   VAR
      s_FB_TimerOnOffDelay_Connected { ExternalAccessible := 'False'; ExternalVisible := 'False'; ExternalWritable := 'False'; S7_SetPoint := 'False'} : "FB_TimerOnOffDelay";
      sR_TRIG_LogOffRequest {InstructionName := 'R_TRIG'; LibVersion := '1.0'; ExternalAccessible := 'False'; ExternalVisible := 'False'; ExternalWritable := 'False'; S7_SetPoint := 'False'} : R_TRIG;   // Siemens "R_TRIG" - to prepare the rising edge trigger on "ix_LogOffRequest" signal
      sUDT_MessageArray { ExternalAccessible := 'False'; ExternalVisible := 'False'; ExternalWritable := 'False'; S7_SetPoint := 'False'} : "UDT_Message";   // Message character array
      sa_Status { ExternalAccessible := 'False'; ExternalVisible := 'False'; ExternalWritable := 'False'} : Struct   // Status structure
         FIFOStatus { ExternalAccessible := 'False'; ExternalVisible := 'False'; ExternalWritable := 'False'} : "UDT_FifoStatus";   // FIFO status structure
         FIFOError { ExternalAccessible := 'False'; ExternalVisible := 'False'; ExternalWritable := 'False'; S7_SetPoint := 'True'} : Bool;   // FIFO data buffer full
         FIFOWarning { ExternalAccessible := 'False'; ExternalVisible := 'False'; ExternalWritable := 'False'; S7_SetPoint := 'True'} : Bool;   // FIFO Warning
         InvalidMsgArraySize { ExternalAccessible := 'False'; ExternalVisible := 'False'; ExternalWritable := 'False'} : Bool;   // Invalig message array size
      END_STRUCT;
      ss_Message { ExternalAccessible := 'False'; ExternalVisible := 'False'; ExternalWritable := 'False'} : String;   // Message character string
      sui_MsgArrayElNr { ExternalAccessible := 'False'; ExternalVisible := 'False'; ExternalWritable := 'False'} : UInt;   // Invalid message array size
      si_MaxMsgLen { ExternalAccessible := 'False'; ExternalVisible := 'False'; ExternalWritable := 'False'} : Int;   // Maximum message length
      si_MsgLen { ExternalAccessible := 'False'; ExternalVisible := 'False'; ExternalWritable := 'False'} : Int;   // String character message length
   END_VAR

   VAR CONSTANT
      cc_NULL : Char := '$00';   // NULL sign
      cc_STX : Char := '$02';   // Start of the text
      cc_ETX : Char := '$03';   // End of the text
      cs_MessageLength : String := '0006';   // Legth of the message
      cs_LogOffRequest : String := 'LS';   // Message type
   END_VAR


BEGIN
	(*
	----------------------------------------------------------------------------------------

	Version history:
	Date        | Version   | Author        | Remark
	----------------------------------------------------------------------------------------
	24/05/2019  | 0.1       | L.Klar        | first release MHS TIA 15.1
	29/06/2021  | 1.0       | F.Baten       | first release MHS TIA 16.4
	08/11/2021  | 1.1       | M.Piela       | Interface changes
	05/04/2022  | 1.2       | K.Pokorski    | Review
	21/02/2023  | 4.0       | F.Baten       | 4.0 Release TIA 17.5
	*)

	REGION 1 – FIFO header status update

	    // Mode 'S' - FIFO register status update
	    "FC_Fifo"(ic_Mode := 'S',
	              qUDT_Status => #sa_Status.FIFOStatus,
	              qx_Error => #sa_Status.FIFOError,
	              qx_Warning => #sa_Status.FIFOWarning,
	              iqv_Data := #sUDT_MessageArray,
	              iqUDT_FifoHeader := #iqUDT_FifoHeader,
	              iqv_DataBuffer := #iqa_FifoData);

	END_REGION

	REGION 2 – Message preparation

	    #s_FB_TimerOnOffDelay_Connected(iudi_OnDelayTime := #i_UDT_Facility_PLC.SS,
	                                    iudi_OffDelayTime := 0,
	                                    ix_SignalToDelay := #ix_Connected AND NOT #ix_ConnectionAccepted);


	    #sR_TRIG_LogOffRequest(CLK := #ix_LogOffRequest OR #s_FB_TimerOnOffDelay_Connected.qx_DelayedSignal);

	    IF (NOT #iqUDT_FifoHeader.Status.Full)                 // FIFO isn't full
	    THEN

	        IF (#sR_TRIG_LogOffRequest.Q                       // Trigger message
	            AND NOT #sa_Status.FIFOError)                   // No FIFO error
	        THEN
	            REGION 2.1 – Message preparation

	                // Heartbeat message composing according to the structure: STX,00,06,LS,ETX
	                #ss_Message := CONCAT(IN1 := #cc_STX,             // Start of message
	                                      IN2 := #cs_MessageLength,            // message length
	                                      IN3 := #cs_LogOffRequest,     // Log-off request message
	                                      IN4 := #cc_ETX);              // End of message

	            END_REGION

	            REGION 2.2 – Maximum number of the message characters

	                #si_MaxMsgLen := "FC_GetNrOfArrayEl"(iv_Array := #sUDT_MessageArray.Character);

	            END_REGION

	            REGION 2.3 – Length of the complete message

	                #si_MsgLen := LEN(#ss_Message);

	            END_REGION

	            REGION 2.4 –  Message array size validation

	                #sa_Status.InvalidMsgArraySize := #si_MsgLen > #si_MaxMsgLen;

	            END_REGION

	            REGION 2.5 –  Message character string conversion to a message array of characters

	                IF (NOT #sa_Status.InvalidMsgArraySize)     // Message character array size is valid
	                THEN

	                    Strg_TO_Chars(Strg := #ss_Message,
	                                  pChars := 0,
	                                  Cnt => #sui_MsgArrayElNr,
	                                  Chars := #sUDT_MessageArray.Character);
	                END_IF;

	            END_REGION

	            REGION 2.6 – Clearing remaining characters in the message character array

	                IF (NOT #sa_Status.InvalidMsgArraySize)     // Message character array size is valid
	                THEN

	                    // Filling up not used message character array elements with '$00' (ASCII - 16#00)
	                    FILL_BLK(IN := #cc_NULL,
	                             COUNT := UINT_TO_ULINT(INT_TO_UINT(#si_MaxMsgLen) - #sui_MsgArrayElNr),
	                             OUT => #sUDT_MessageArray.Character[#sui_MsgArrayElNr]);

	                END_IF;

	            END_REGION

	            REGION 2.7 – Message write into a FIFO register

	                IF NOT #sa_Status.InvalidMsgArraySize // Message character array size is valid
	                THEN

	                    // Mode 'W' - Write FIFO record
	                    "FC_Fifo"(ic_Mode := 'W',
	                              qUDT_Status => #sa_Status.FIFOStatus,
	                              qx_Error => #sa_Status.FIFOError,
	                              qx_Warning => #sa_Status.FIFOWarning,
	                              iqv_Data := #sUDT_MessageArray,
	                              iqUDT_FifoHeader := #iqUDT_FifoHeader,
	                              iqv_DataBuffer := #iqa_FifoData);
	                END_IF;

	            END_REGION

	        END_IF;

	        // In case of FIFO full, the FIFO full error bit and FIFO collective error bit are set
	    ELSE

	        #sa_Status.FIFOError := TRUE;
	        #sa_Status.FIFOStatus.FifoFull := TRUE;

	    END_IF;

	END_REGION

	REGION Close connection

	    IF #iqUDT_FifoHeader.TotalEntriesStored = 0
	        AND (#ix_LogOffRequest OR #s_FB_TimerOnOffDelay_Connected.qx_DelayedSignal)
	    THEN
	        #iqx_Reconnect := TRUE;
	    END_IF;


	END_REGION


	REGION 3 - Writing output

	    #qx_Error := #sa_Status.InvalidMsgArraySize         // Invalid message array size
	    OR #sa_Status.FIFOError;                            // FIFO error

	END_REGION
END_FUNCTION_BLOCK

FUNCTION_BLOCK "FB_FedExPacketLengthMessage"
TITLE = FB_Heartbeat
{ S7_Optimized_Access := 'TRUE' }
AUTHOR : MHSE
FAMILY : UPS_SpecificCommunication
VERSION : 3.0
// ATTRIBUTES
// AUTO_NUMBER = True
// BLOCK_NUMBER = 80
// END_ATTRIBUTES
//Function block to send and monitor the UPS heartbeat message.
   VAR_INPUT
      iUDT_Facility { ExternalAccessible := 'False'; ExternalVisible := 'False'; ExternalWritable := 'False'} : "UDT_FedExFacility";   // System configuration
      is_LOConEquipment { ExternalAccessible := 'False'; ExternalVisible := 'False'; ExternalWritable := 'False'} : String[3];   // Location of the equipment
      is_DEPCOD { ExternalAccessible := 'False'; ExternalVisible := 'False'; ExternalWritable := 'False'} : String[6];   // Depot Code
      is_TYPofEquipment { ExternalAccessible := 'False'; ExternalVisible := 'False'; ExternalWritable := 'False'} : String[3];   // Type of equipment
      is_NumberOfTheEquipment { ExternalAccessible := 'False'; ExternalVisible := 'False'; ExternalWritable := 'False'} : String[3];   // Number of the equipment 001-999
      is_TrayCellNumber { ExternalAccessible := 'False'; ExternalVisible := 'False'; ExternalWritable := 'False'} : String[3];   // Tray/Cell number (for loop sorters) or generated by LLC (on line sorters).
      is_SorterNumber { ExternalAccessible := 'False'; ExternalVisible := 'False'; ExternalWritable := 'False'} : String[2];   // Sorter number
      is_InductionNumber { ExternalAccessible := 'False'; ExternalVisible := 'False'; ExternalWritable := 'False'} : String[2];   // Induction number
      is_AreaNumber { ExternalAccessible := 'False'; ExternalVisible := 'False'; ExternalWritable := 'False'} : String[2];   // Area number
      ii_Gin { ExternalAccessible := 'False'; ExternalVisible := 'False'; ExternalWritable := 'False'} : Int;   // GIN number
   END_VAR

   VAR_OUTPUT
      qx_Error { ExternalAccessible := 'False'; ExternalVisible := 'False'; ExternalWritable := 'False'} : Bool;   // Error
   END_VAR

   VAR_IN_OUT
      iqUDT_FifoHeader : "UDT_FifoHeader";   // FIFO header
      iqa_FifoData : Array[*] of "UDT_Message";   // FIFO data
      iqUDT_CustomerID : "UDT_FedExCustomerID";
   END_VAR

   VAR
      sFB_FedExCustomerID { ExternalAccessible := 'False'; ExternalVisible := 'False'; ExternalWritable := 'False'; S7_SetPoint := 'False'} : "FB_FedExCustomerID";
      sUDT_MessageArray { ExternalAccessible := 'False'; ExternalVisible := 'False'; ExternalWritable := 'False'; S7_SetPoint := 'False'} : "UDT_Message";   // Message character array
      sa_Status { ExternalAccessible := 'False'; ExternalVisible := 'False'; ExternalWritable := 'False'} : Struct   // Status structure
         FIFOStatus { ExternalAccessible := 'False'; ExternalVisible := 'False'; ExternalWritable := 'False'} : "UDT_FifoStatus";   // FIFO status structure
         FIFOError { ExternalAccessible := 'False'; ExternalVisible := 'False'; ExternalWritable := 'False'; S7_SetPoint := 'True'} : Bool;   // FIFO data buffer full
         FIFOWarning { ExternalAccessible := 'False'; ExternalVisible := 'False'; ExternalWritable := 'False'; S7_SetPoint := 'True'} : Bool;   // FIFO error
         InvalidGIN { ExternalAccessible := 'False'; ExternalVisible := 'False'; ExternalWritable := 'False'} : Bool;   //  Invalid GIN
         InvalidMessageLength { ExternalAccessible := 'False'; ExternalVisible := 'False'; ExternalWritable := 'False'} : Bool;   // Calculated message length is different than required
         InvalidMsgArraySize { ExternalAccessible := 'False'; ExternalVisible := 'False'; ExternalWritable := 'False'} : Bool;   // Length of the message is bigger than length of message array
      END_STRUCT;
      sa_Statistics { ExternalAccessible := 'False'; ExternalVisible := 'False'; ExternalWritable := 'False'} : Struct   // Statistics structure
         NotSentWrongMsgLen { ExternalAccessible := 'False'; ExternalVisible := 'False'; ExternalWritable := 'False'} : DInt;   // COMISSIONING PURPOSE Messages not sent because built message length does not match with required message length
      END_STRUCT;
      ss_LLCSystemID { ExternalAccessible := 'False'; ExternalVisible := 'False'; ExternalWritable := 'False'} : String[15];   // Identifier of Low-Level controls
      ss_SequencialID { ExternalAccessible := 'False'; ExternalVisible := 'False'; ExternalWritable := 'False'} : String[6];   // Identifier of Low-Level controls
      ss_Message { ExternalAccessible := 'False'; ExternalVisible := 'False'; ExternalWritable := 'False'} : String;   // Message character string
      ss_PackageID { ExternalAccessible := 'False'; ExternalVisible := 'False'; ExternalWritable := 'False'} : String;   // Identifier of Low-Level controls
      ss_LEN { ExternalAccessible := 'False'; ExternalVisible := 'False'; ExternalWritable := 'False'} : String;   // Length of message
      ss_Gap { ExternalAccessible := 'False'; ExternalVisible := 'False'; ExternalWritable := 'False'} : String;   // Parcel leading gap
      ss_GapUOM { ExternalAccessible := 'False'; ExternalVisible := 'False'; ExternalWritable := 'False'} : String;   // Gap units
      ss_Length { ExternalAccessible := 'False'; ExternalVisible := 'False'; ExternalWritable := 'False'} : String;   // Parcel length
      sui_MsgArrayElNr { ExternalAccessible := 'False'; ExternalVisible := 'False'; ExternalWritable := 'False'} : UInt;   // Message array size
      si_OldGin { ExternalAccessible := 'False'; ExternalVisible := 'False'; ExternalWritable := 'False'} : Int;   // Previous Gin
      si_StringLen { ExternalAccessible := 'False'; ExternalVisible := 'False'; ExternalWritable := 'False'} : Int;   // Length of string used in loops to pad string with spaces or 0
      si_LenFillLoop { ExternalAccessible := 'False'; ExternalVisible := 'False'; ExternalWritable := 'False'} : Int;   // Loop couter
      si_MaxMsgLen { ExternalAccessible := 'False'; ExternalVisible := 'False'; ExternalWritable := 'False'} : Int;   // Maximum message length
      si_MsgLen { ExternalAccessible := 'False'; ExternalVisible := 'False'; ExternalWritable := 'False'} : Int;   // String character message length
   END_VAR

   VAR CONSTANT
      cc_NULL : Char := '$00';   // NULL sign
      cc_STX : Char := '$02';   // Start of the text
      cc_ETX : Char := '$03';   // End of the text
      cs_Length : String := '0081';   // Legth of the message
      cs_MessageType : String := 'PL';   // Message type
   END_VAR


BEGIN
	(*
	----------------------------------------------------------------------------------------

	Version history:
	Date        | Version   | Author        | Remark
	----------------------------------------------------------------------------------------
	29/06/2021  | 1.0       | F.Baten       | first release MHS TIA 16.0
	10/11/2021  | 1.2       | M.Piela       | Updating regions numbering and interface changes
	05/04/2022  | 1.3       | K.Pokorski    | Review
	30/06/2022  | 1.4       | K.Pokorski    | Add cusotmer ID generation and swap GIN with Customer ID
	21/02/2023  | 4.0       | F.Baten       | 4.0 Release TIA 17.5
	*)

	REGION 1 – FIFO header status update

	    // Mode 'S' - FIFO register status update
	    "FC_Fifo"(ic_Mode := 'S',
	              qUDT_Status => #sa_Status.FIFOStatus,
	              qx_Error => #sa_Status.FIFOError,
	              qx_Warning => #sa_Status.FIFOWarning,
	              iqv_Data := #sUDT_MessageArray,
	              iqUDT_FifoHeader := #iqUDT_FifoHeader,
	              iqv_DataBuffer := #iqa_FifoData);
	END_REGION

	REGION 2 - GIN validation

	    // GIN validation
	    #sa_Status.InvalidGIN :=
	    #ii_Gin < 1
	    OR #ii_Gin > 9999;

	END_REGION

	REGION 3 – Message preparation

	    IF NOT #iqUDT_FifoHeader.Status.Full                 // FIFO isn't full
	    THEN
	        IF #ii_Gin <> #si_OldGin AND NOT #sa_Status.InvalidGIN

	        THEN
	            REGION 3.1 - Sequencial ID

	                // Assign CustomerID
	                #sFB_FedExCustomerID(ii_Gin := #ii_Gin,
	                                     iqUDT_CustomerID := #iqUDT_CustomerID);


	                // ss_SequencialID character string clearing
	                #ss_SequencialID := '';

	                // ss_SequencialID double integer input conversion to a character string
	                VAL_STRG(IN := "DB_GIN".GIN[#ii_Gin].FedEx.CustomerID,
	                         SIZE := 0,
	                         PREC := 0,
	                         FORMAT := 0,
	                         P := 1,
	                         OUT => #ss_SequencialID);
	                // Length of the ss_SequencialID character string
	                #si_StringLen := LEN(#ss_SequencialID);

	                // ss_SequencialID character string leading zeros addition
	                IF (#si_StringLen < 6)
	                THEN
	                    FOR #si_LenFillLoop := 1 TO 6 - #si_StringLen DO
	                        #ss_SequencialID := CONCAT(IN1 := '0',
	                                                   IN2 := #ss_SequencialID);
	                    END_FOR;
	                END_IF;
	            END_REGION

	            REGION 3.2 - LLC System ID
	                // Build LLC Syatem ID
	                #ss_LLCSystemID := CONCAT(IN1 := #is_DEPCOD,
	                                          IN2 := #is_LOConEquipment,
	                                          IN3 := #is_TYPofEquipment,
	                                          IN4 := #is_NumberOfTheEquipment);
	            END_REGION

	            REGION 3.3 - Package ID
	                // Build Package ID
	                #ss_PackageID := CONCAT(IN1 := #is_TrayCellNumber,
	                                        IN2 := #is_SorterNumber,
	                                        IN3 := #is_InductionNumber,
	                                        IN4 := #is_AreaNumber,
	                                        IN5 := #ss_SequencialID);
	            END_REGION

	            REGION 3.4 - Gap
	                // Gap character string clearing
	                #ss_Gap := '';

	                IF ("DB_GIN".GIN[#ii_Gin].General.LeadingGap > 999)
	                THEN
	                    #ss_Gap := '999';
	                ELSE

	                    // Gap integer input conversion to a character string
	                    VAL_STRG(IN := "DB_GIN".GIN[#ii_Gin].General.LeadingGap,
	                             SIZE := 0,
	                             PREC := 0,
	                             FORMAT := 0,
	                             P := 1,
	                             OUT => #ss_Gap);
	                    // Length of the gap character string
	                    #si_StringLen := LEN(#ss_Gap);
	                    // Gap character string leading zeros addition
	                    IF (#si_StringLen < 3)
	                    THEN
	                        FOR #si_LenFillLoop := 1 TO 3 - #si_StringLen DO
	                            #ss_Gap := CONCAT(IN1 := '0',
	                                              IN2 := #ss_Gap);
	                        END_FOR;
	                    END_IF;
	                END_IF;
	                #ss_GapUOM := 'CM';
	            END_REGION

	            REGION 3.5 - Length
	                // Length character string clearing
	                #ss_Length := '';
	                // Gap integer input conversion to a character string
	                VAL_STRG(IN := "DB_GIN".GIN[#ii_Gin].General.Length,
	                         SIZE := 0,
	                         PREC := 0,
	                         FORMAT := 0,
	                         P := 1,
	                         OUT => #ss_Length);
	                // Length of the gap character string
	                #si_StringLen := LEN(#ss_Length);
	                // Gap character string leading zeros addition
	                IF (#si_StringLen < 3)
	                THEN
	                    FOR #si_LenFillLoop := 1 TO 3 - #si_StringLen DO
	                        #ss_Length := CONCAT(IN1 := '0',
	                                             IN2 := #ss_Length);
	                    END_FOR;
	                END_IF;

	            END_REGION


	            REGION 3.6 – Message preparation
	                // Message composing according to the structure: STX,BODY ,ETX
	                #ss_Message := CONCAT(IN1 := #cc_STX,
	                                      IN2 := #cs_Length,
	                                      IN3 := #cs_MessageType,
	                                      IN4 := #ss_LLCSystemID,
	                                      IN5 := #ss_PackageID,
	                                      IN6 := "DB_GIN".GIN[#ii_Gin].FedEx.PackageEntrancePoint,
	                                      IN7 := "DB_GIN".GIN[#ii_Gin].FedEx.PackageEntranceState,
	                                      IN8 := #ss_Gap,
	                                      IN9 := #ss_Length,
	                                      IN10 := #ss_GapUOM,
	                                      IN11 := "DB_Time".Timestamp,
	                                      IN12 := #iUDT_Facility.TimeZoneDesignator,
	                                      IN13 := #cc_ETX);

	            END_REGION

	            REGION 3.7 – Maximum number of the message characters

	                #si_MaxMsgLen := "FC_GetNrOfArrayEl"(iv_Array := #sUDT_MessageArray.Character);

	            END_REGION

	            REGION 3.8 – Length of the complete message

	                #si_MsgLen := LEN(#ss_Message);

	                // Message length validation
	                #sa_Status.InvalidMessageLength := #si_MsgLen - 2 <> STRING_TO_INT(#cs_Length);

	            END_REGION

	            REGION 3.9 –  Message array size validation

	                #sa_Status.InvalidMsgArraySize := #si_MsgLen > #si_MaxMsgLen;

	            END_REGION

	            REGION 3.10 –  Message character string conversion to a message array of characters

	                IF (NOT #sa_Status.InvalidMsgArraySize)     // Message character array size is valid
	                THEN

	                    Strg_TO_Chars(Strg := #ss_Message,
	                                  pChars := 0,
	                                  Cnt => #sui_MsgArrayElNr,
	                                  Chars := #sUDT_MessageArray.Character);

	                END_IF;

	            END_REGION

	            REGION 3.11 – Clearing remaining characters in the message character array

	                IF (NOT #sa_Status.InvalidMsgArraySize)     // Message character array size is valid
	                THEN

	                    // Filling up not used message character array elements with '$00' (ASCII - 16#00)
	                    FILL_BLK(IN := #cc_NULL,
	                             COUNT := UINT_TO_ULINT(INT_TO_UINT(#si_MaxMsgLen) - #sui_MsgArrayElNr),
	                             OUT => #sUDT_MessageArray.Character[#sui_MsgArrayElNr]);

	                END_IF;

	            END_REGION

	            REGION 3.12 – Message write into a FIFO register

	                IF NOT #sa_Status.InvalidMsgArraySize          // Message character array size is valid
	                    AND NOT #sa_Status.InvalidMessageLength     // Message length size validation
	                THEN

	                    // Mode 'W' - Write FIFO record
	                    "FC_Fifo"(ic_Mode := 'W',
	                              qUDT_Status => #sa_Status.FIFOStatus,
	                              qx_Error => #sa_Status.FIFOError,
	                              qx_Warning => #sa_Status.FIFOWarning,
	                              iqv_Data := #sUDT_MessageArray,
	                              iqUDT_FifoHeader := #iqUDT_FifoHeader,
	                              iqv_DataBuffer := #iqa_FifoData);
	                ELSE
	                    // Increase counter messages not sent because of wrong message length
	                    #sa_Statistics.NotSentWrongMsgLen += 1;


	                END_IF;

	            END_REGION
	            #si_OldGin := #ii_Gin;
	        END_IF;
	        // In case of FIFO full, the FIFO full error bit and FIFO collective error bit are set
	    ELSE

	        #sa_Status.FIFOError := TRUE;
	        #sa_Status.FIFOStatus.FifoFull := TRUE;

	    END_IF;

	END_REGION

	REGION 4 - Writing outputs

	    #qx_Error := #sa_Status.InvalidMessageLength        // Invalid message length
	    OR #sa_Status.InvalidGIN                            // Invalid GIN
	    OR #sa_Status.InvalidMsgArraySize                   // Invalid message array size
	    OR #sa_Status.FIFOError;                            // FIFO error

	END_REGION
END_FUNCTION_BLOCK

FUNCTION_BLOCK "FB_FedExChute2Brakes1Stop"
{ S7_Optimized_Access := 'TRUE' }
VERSION : 0.1
// ATTRIBUTES
// AUTO_NUMBER = True
// BLOCK_NUMBER = 237
// END_ATTRIBUTES
   VAR_INPUT
      iUDT_ChuteConfiguration { ExternalAccessible := 'False'; ExternalVisible := 'False'; ExternalWritable := 'False'} : "UDT_Chute3BrakesConfiguration";   // Chute configuration structure
      iUDT_Facility { ExternalAccessible := 'False'; ExternalVisible := 'False'; ExternalWritable := 'False'} : "UDT_FedExFacility";   // System configuration
      ix_PECChuteFull { ExternalAccessible := 'False'; ExternalVisible := 'False'; ExternalWritable := 'False'} : Bool;   // TRUE when chute full photoye is not blocked
      ix_PECBrakeTop { ExternalAccessible := 'False'; ExternalVisible := 'False'; ExternalWritable := 'False'} : Bool;   // TRUE when first (Top) brake assembly photoye is not blocked
      ix_PECBrakeMiddle { ExternalAccessible := 'False'; ExternalVisible := 'False'; ExternalWritable := 'False'} : Bool;   // TRUE when second (Middle) brake assembly photoye is not blocked
      ix_PECBrakeBottom { ExternalAccessible := 'False'; ExternalVisible := 'False'; ExternalWritable := 'False'} : Bool;   // TRUE when third (End Stop) brake assembly photoye is not blocked
      ix_PECStopTop { ExternalAccessible := 'False'; ExternalVisible := 'False'; ExternalWritable := 'False'} : Bool;   // TRUE when first/Top brake assembly photoye is not blocked
      ix_PECStopMiddle { ExternalAccessible := 'False'; ExternalVisible := 'False'; ExternalWritable := 'False'} : Bool;   // TRUE when second/Middle brake assembly photoye is not blocked
      ix_PECStopBottom { ExternalAccessible := 'False'; ExternalVisible := 'False'; ExternalWritable := 'False'} : Bool;   // TRUE when third/(End Stop) brake assembly photoye is not blocked
      ix_ChuteJam { ExternalAccessible := 'False'; ExternalVisible := 'False'; ExternalWritable := 'False'} : Bool;   // TRUE when external jam appear
      ix_SafetyOk { ExternalAccessible := 'False'; ExternalVisible := 'False'; ExternalWritable := 'False'} : Bool;   // TRUE when safety is ok
      ix_HardwareOk { ExternalAccessible := 'False'; ExternalVisible := 'False'; ExternalWritable := 'False'} : Bool;   // TRUE when hardware is ok
      ix_EnergySave { ExternalAccessible := 'False'; ExternalVisible := 'False'; ExternalWritable := 'False'} : Bool;   // TRUE when enery save is active
   END_VAR

   VAR_OUTPUT
      qUDT_HMIStatus { ExternalAccessible := 'False'; ExternalVisible := 'False'; ExternalWritable := 'False'} : "UDT_Chute3BrakeStatus";   // HMI status structure
      qUDT_Status { ExternalAccessible := 'False'; ExternalVisible := 'False'; ExternalWritable := 'False'} : "UDT_CommonStatus";   // Common status structure
      qUDT_StatusToXBS { ExternalAccessible := 'False'; ExternalVisible := 'False'; ExternalWritable := 'False'} : "UDT_XBSChuteInterfaceSend";
      qx_Lamp { ExternalAccessible := 'False'; ExternalVisible := 'False'; ExternalWritable := 'False'} : Bool;   // Chute Lamp Jam/Full
      qx_BrakeValve1 { ExternalAccessible := 'False'; ExternalVisible := 'False'; ExternalWritable := 'False'} : Bool;   // First brake valve assembly
      qx_BrakeValve2 { ExternalAccessible := 'False'; ExternalVisible := 'False'; ExternalWritable := 'False'} : Bool;   // Second brake valve  assembly
      qx_BrakeValve3 { ExternalAccessible := 'False'; ExternalVisible := 'False'; ExternalWritable := 'False'} : Bool;   // Third brake valve assembly
   END_VAR

   VAR_IN_OUT
      iqUDT_EquipmentControl : "UDT_EquipmentControl";   // Equipment control structure
      iqUDT_Statistics : "UDT_Chute3BrakeStatistics";   // Statistics structure
      iqUDT_HandShake : "UDT_ConveyorHandshake";   // Downstream handshake structure
      iqUDT_HandShakeUp : "UDT_ConveyorHandshake";   // Upstream handshake structure
      iqUDT_ChuteCommand : "UDT_Chute3BrakeCommand";   // Command strucutre
      iqUDT_FifoHighPriorityHLC : "UDT_FifoHeader";   // FIFO UDS send Header
      iqa_FifoHighPriorityHLC : Array[*] of "UDT_Message";   // FIFO UDS send data
   END_VAR

   VAR
      sUDT_CommonStatus { ExternalAccessible := 'False'; ExternalVisible := 'False'; ExternalWritable := 'False'; S7_SetPoint := 'False'} : "UDT_CommonStatus";   // Common status structure
      sUDT_CommonStatusOld { ExternalAccessible := 'False'; ExternalVisible := 'False'; ExternalWritable := 'False'; S7_SetPoint := 'False'} : "UDT_CommonStatus";   // Auxiliary status structure
      sUDT_HMIStatus { ExternalAccessible := 'False'; ExternalVisible := 'False'; ExternalWritable := 'False'; S7_SetPoint := 'False'} : "UDT_Chute3BrakeStatus";   // HMI status structure
      sUDT_Configuration { ExternalAccessible := 'False'; ExternalVisible := 'False'; ExternalWritable := 'False'; S7_SetPoint := 'False'} : "UDT_Chute3BrakesConfiguration";   // Auxiliary equipment control structure
      sFB_PneumaticBrakeUnitAssemby1 { ExternalAccessible := 'False'; ExternalVisible := 'False'; ExternalWritable := 'False'; S7_SetPoint := 'False'} : "FB_PneumaticBrakeUnit";   // Function to control a first pneumatic brake contol
      sFB_PneumaticBrakeUnitAssemby2 { ExternalAccessible := 'False'; ExternalVisible := 'False'; ExternalWritable := 'False'; S7_SetPoint := 'False'} : "FB_PneumaticBrakeUnit";   // Function to control a secound pneumatic brake contol
      sFB_StopRoller { ExternalAccessible := 'False'; ExternalVisible := 'False'; ExternalWritable := 'False'; S7_SetPoint := 'False'} : "FB_StopRoller";   // Function to control stoping of the roller
      sFB_FedExEquipmentStatusMessage { ExternalAccessible := 'False'; ExternalVisible := 'False'; ExternalWritable := 'False'; S7_SetPoint := 'False'} : "FB_FedExEquipmentStatusMessage";   // Equipment status structure message
      sFB_TimerOnOffDelayPECFul { ExternalAccessible := 'False'; ExternalVisible := 'False'; ExternalWritable := 'False'; S7_SetPoint := 'False'} : "FB_TimerOnOffDelay";   // Filtering full photo eye signal
      sFB_TimerOnOffDelayPECHalfFull { ExternalAccessible := 'False'; ExternalVisible := 'False'; ExternalWritable := 'False'; S7_SetPoint := 'False'} : "FB_TimerOnOffDelay";   // Filtering half full photo eye signal
      sFB_TimerOnOffDelayPECMiddle { ExternalAccessible := 'False'; ExternalVisible := 'False'; ExternalWritable := 'False'; S7_SetPoint := 'False'} : "FB_TimerOnOffDelay";   // Filtering middle photo eye signal
      sFB_TimerOnOffDelayStopRollerLongBrakePause { ExternalAccessible := 'False'; ExternalVisible := 'False'; ExternalWritable := 'False'; S7_SetPoint := 'False'} : "FB_TimerOnOffDelay";   // Filtering common signal from all signals needed to increase brake pause
      sR_TRIG_ChuteFull {InstructionName := 'R_TRIG'; LibVersion := '1.0'; ExternalAccessible := 'False'; ExternalVisible := 'False'; ExternalWritable := 'False'; S7_SetPoint := 'False'} : R_TRIG;   // Rising edge to chute full
      sR_TRIG_ChuteJam {InstructionName := 'R_TRIG'; LibVersion := '1.0'; ExternalAccessible := 'False'; ExternalVisible := 'False'; ExternalWritable := 'False'; S7_SetPoint := 'False'} : R_TRIG;   // Rising edge to chute jam
      sR_TRIG_ChuteHalfFull {InstructionName := 'R_TRIG'; LibVersion := '1.0'; ExternalAccessible := 'False'; ExternalVisible := 'False'; ExternalWritable := 'False'; S7_SetPoint := 'False'} : R_TRIG;   // Rising edge to chute half full
      sR_TRIG_DisableFromHMI {InstructionName := 'R_TRIG'; LibVersion := '1.0'; ExternalAccessible := 'False'; ExternalVisible := 'False'; ExternalWritable := 'False'; S7_SetPoint := 'False'} : R_TRIG;   // Rising edge to disable chute from HMI
      sR_TRIG_DisableFromHLC {InstructionName := 'R_TRIG'; LibVersion := '1.0'; ExternalAccessible := 'False'; ExternalVisible := 'False'; ExternalWritable := 'False'; S7_SetPoint := 'False'} : R_TRIG;   // Rising edge to disable chute from HLC
      sF_TRIG_UpdateStatus {InstructionName := 'F_TRIG'; LibVersion := '1.0'; ExternalAccessible := 'False'; ExternalVisible := 'False'; ExternalWritable := 'False'; S7_SetPoint := 'False'} : F_TRIG;
      ss_StatusCode { ExternalAccessible := 'False'; ExternalVisible := 'False'; ExternalWritable := 'False'} : String[3];   // Status code
      sx_MasterValve { ExternalAccessible := 'False'; ExternalVisible := 'False'; ExternalWritable := 'False'} : Bool;   // Master valve
      sx_StopActive1 { ExternalAccessible := 'False'; ExternalVisible := 'False'; ExternalWritable := 'False'} : Bool;   // First brake valve assembly is active
      sx_StopActive2 { ExternalAccessible := 'False'; ExternalVisible := 'False'; ExternalWritable := 'False'} : Bool;   // Second brake valve assembly is active
      sx_StopActive3 { ExternalAccessible := 'False'; ExternalVisible := 'False'; ExternalWritable := 'False'} : Bool;   // Third brake valve assembly is active
      sx_PECFullFiltered { ExternalAccessible := 'False'; ExternalVisible := 'False'; ExternalWritable := 'False'} : Bool;   // Delayed full photo eye signal
      sx_PECHalfFullFiltered { ExternalAccessible := 'False'; ExternalVisible := 'False'; ExternalWritable := 'False'} : Bool;   // Delayed half full photo eye signal
      sx_PECMiddleFullFiltered { ExternalAccessible := 'False'; ExternalVisible := 'False'; ExternalWritable := 'False'} : Bool;   // Delayed middle full photo eye signal
      sx_StopRollerLongBrakePauseDelayed { ExternalAccessible := 'False'; ExternalVisible := 'False'; ExternalWritable := 'False'} : Bool;   // Delayed common signal from all signals needed to increase brake pause
      sx_StopRollerLongBrakePause { ExternalAccessible := 'False'; ExternalVisible := 'False'; ExternalWritable := 'False'} : Bool;   // Common signal from all signals needed to increase brake pause
      sx_ChuteFull { ExternalAccessible := 'False'; ExternalVisible := 'False'; ExternalWritable := 'False'} : Bool;   // Full status
      sx_ChuateHalfFull { ExternalAccessible := 'False'; ExternalVisible := 'False'; ExternalWritable := 'False'} : Bool;   // Half full occupation status
      sx_ChuteJam { ExternalAccessible := 'False'; ExternalVisible := 'False'; ExternalWritable := 'False'} : Bool;   // Jam status
      sx_MessageError { ExternalAccessible := 'False'; ExternalVisible := 'False'; ExternalWritable := 'False'} : Bool;   // Message error
   END_VAR


BEGIN
	(*
	----------------------------------------------------------------------------------------

	Version history:
	Date        | Version   | Author        | Remark
	----------------------------------------------------------------------------------------
	23/06/2021  | 0.0       | F. Baten      | first release TIA 15.1
	20/10/2021  | 0.1       | M. Piela      | Add statuses and statistics. Stylistic correction
	21/10/2021  | 0.2       | M. Piela      | Change brake stopper pause based on all pec delayed signal
	02/02/2022  | 0.3       | M. Piela      | Add Equipment status message
	22/02/2022  | 0.4       | M. Piela      | Update HMI Status
	04/04/2022  | 0.5       | S. Deulkar    | Updated status for XBS sorter
	25/06/2022  | 0.6       | M. Kurpiers   | Interface update
	25/06/2022  | 0.7       | M. Piela      | #sx_MasterValve inverted to top brake
	19/07/2022  | 0.8       | M. Piela      | Add external chute jam to the status
	21/02/2023  | 4.0       | F.Baten       | 4.0 Release TIA 17.5
	 *)

	REGION 1 - Write input status

	    IF #ix_HardwareOk
	    THEN
	        #sUDT_HMIStatus.Specific.DisableFromHMI := #iqUDT_ChuteCommand.DisableFromHMI;
	        #sUDT_HMIStatus.Specific.DisableFromHLC := #iqUDT_ChuteCommand.DisableFromHLC;
	        #sUDT_HMIStatus.Specific.ChuteFull := #sx_ChuteFull;
	        #sUDT_HMIStatus.Specific.ChuteHalfFull := #sx_ChuateHalfFull;
	        #sUDT_HMIStatus.Specific.ChuteJam := #sx_ChuteJam OR #ix_ChuteJam;
	        #sUDT_HMIStatus.Specific.BrakeFaultTop := FALSE;
	        #sUDT_HMIStatus.Specific.BrakeFaultMiddle := FALSE;
	        #sUDT_HMIStatus.Specific.BrakeFaultBottom := FALSE;
	    END_IF;

	END_REGION

	REGION 2 - Triggers

	    // Rising edge trigger full PEC status
	    #sR_TRIG_ChuteFull(CLK := #sx_ChuteFull);

	    // Rissing edge trigger jam PEC status
	    #sR_TRIG_ChuteJam(CLK := #sx_ChuteJam);

	    // Rissing edge trigger hafl full PEC status
	    #sR_TRIG_ChuteHalfFull(CLK := #sx_ChuateHalfFull);

	    // Rising edge trigger disable from HMI
	    #sR_TRIG_DisableFromHMI(CLK := #sUDT_HMIStatus.Specific.DisableFromHMI);

	    // Rising edge trigger disable from MFC
	    #sR_TRIG_DisableFromHLC(CLK := #sUDT_HMIStatus.Specific.DisableFromHLC);

	END_REGION

	REGION 3 - Timers

	    // Filtering full photo eye signal
	    #sFB_TimerOnOffDelayPECFul(iudi_OnDelayTime := #iUDT_ChuteConfiguration.PECFullOnDelay,
	                               iudi_OffDelayTime := #iUDT_ChuteConfiguration.PECFullOffDelay,
	                               ix_SignalToDelay := #ix_PECChuteFull,
	                               ix_Enable := TRUE,
	                               qx_DelayedSignal => #sx_PECFullFiltered);

	    //Filtering Half full photo eye signal
	    #sFB_TimerOnOffDelayPECHalfFull(iudi_OnDelayTime := #iUDT_ChuteConfiguration.PECHalfFullOnDelay,
	                                    iudi_OffDelayTime := #iUDT_ChuteConfiguration.PECHalfFullOffDelay,
	                                    ix_SignalToDelay := #ix_PECStopTop,
	                                    ix_Enable := TRUE,
	                                    qx_DelayedSignal => #sx_PECHalfFullFiltered);

	    //Filtering middle photo eye signal
	    #sFB_TimerOnOffDelayPECMiddle(iudi_OnDelayTime := #iUDT_ChuteConfiguration.PECMiddleOnDelay,
	                                  iudi_OffDelayTime := #iUDT_ChuteConfiguration.PECMiddleOffDelay,
	                                  ix_SignalToDelay := #ix_PECStopMiddle,
	                                  ix_Enable := TRUE,
	                                  qx_DelayedSignal => #sx_PECMiddleFullFiltered);

	    // Create common signal from all signals needed to increase brake pause
	    #sx_StopRollerLongBrakePause := #ix_PECBrakeMiddle
	    AND #ix_PECStopMiddle
	    AND #iqUDT_HandShake.RTR;     // Downstream conveyor is running

	    //Filtering common signal from all signals needed to increase brake pause
	    #sFB_TimerOnOffDelayStopRollerLongBrakePause(iudi_OnDelayTime := #iUDT_ChuteConfiguration.LongBrakePauseOnDelay,
	                                                 ix_SignalToDelay := #sx_StopRollerLongBrakePause,
	                                                 ix_Enable := TRUE,
	                                                 qx_DelayedSignal => #sx_StopRollerLongBrakePauseDelayed);

	END_REGION

	REGION 4 - Brake assembly

	    // Control first pneumatic break unit assembly
	    #sFB_PneumaticBrakeUnitAssemby1(iUDT_PneumaticBreakConfiguration := #iUDT_ChuteConfiguration.BrakeConfiguration1,
	                                    ix_PECBrake := #ix_PECBrakeTop,
	                                    ix_PECStop := #ix_PECStopTop,
	                                    ix_PECdownstream := #ix_PECBrakeMiddle,
	                                    ix_DownstreamStopActive := #sx_StopActive2,
	                                    ix_MasterValve := NOT #sx_MasterValve,
	                                    ix_SafetyOk := #ix_SafetyOk,
	                                    qx_Valve => #qx_BrakeValve1,
	                                    qx_StopActive => #sx_StopActive1,
	                                    iqUDT_EquipmentControl := #iqUDT_EquipmentControl);

	    // Control secound pneumatic break unit assembly
	    #sFB_PneumaticBrakeUnitAssemby2(iUDT_PneumaticBreakConfiguration := #iUDT_ChuteConfiguration.BrakeConfiguration2,
	                                    ix_PECBrake := #ix_PECBrakeMiddle,
	                                    ix_PECStop := #ix_PECStopMiddle,
	                                    ix_PECdownstream := #ix_PECBrakeBottom,
	                                    ix_DownstreamStopActive := #sx_StopActive3,
	                                    ix_SafetyOk := #ix_SafetyOk,
	                                    qx_Valve => #sx_MasterValve,
	                                    qx_StopActive => #sx_StopActive2,
	                                    iqUDT_EquipmentControl := #iqUDT_EquipmentControl);

	    // Control stop roller section
	    #sFB_StopRoller(iUDT_StopRollerConfiguration := #iUDT_ChuteConfiguration.StopperConfiguration,
	                    ix_Pressure := #ix_PECStopMiddle,
	                    ix_PECBrake := #ix_PECBrakeBottom,
	                    ix_PECStop := #ix_PECStopBottom,
	                    ix_DownstreamStopActive := NOT #iqUDT_HandShake.RTR,
	                    ix_SafetyOk := #ix_SafetyOk,
	                    ix_BrakePauseLong := #sx_StopRollerLongBrakePauseDelayed,
	                    qx_Valve => #qx_BrakeValve3,
	                    qx_StopActive => #sx_StopActive3,
	                    iqUDT_EquipmentControl := #iqUDT_EquipmentControl);

	    #qx_BrakeValve2 := #sx_MasterValve;

	END_REGION

	REGION 5 - Filling level

	    //Half full
	    IF NOT #sx_PECMiddleFullFiltered AND NOT #sx_PECHalfFullFiltered
	    THEN
	        #sx_ChuateHalfFull := TRUE;
	    END_IF;
	    IF #sx_PECMiddleFullFiltered AND #sx_PECHalfFullFiltered
	    THEN
	        #sx_ChuateHalfFull := FALSE;
	    END_IF;

	    //Full
	    IF NOT #sx_PECHalfFullFiltered AND NOT #"sx_PECFullFiltered"
	    THEN
	        #sx_ChuteFull := TRUE;
	    END_IF;
	    IF #sx_PECHalfFullFiltered AND #"sx_PECFullFiltered"
	    THEN
	        #sx_ChuteFull := FALSE;
	    END_IF;

	    // Jam
	    #sx_ChuteJam := #sx_PECHalfFullFiltered AND NOT #"sx_PECFullFiltered";

	END_REGION

	REGION 6 - Output

	    //Lamp signal enable
	    #qx_Lamp := NOT (#ix_ChuteJam OR #sx_ChuteJam) AND ((#sx_ChuteFull)
	    OR (#sx_ChuateHalfFull AND "DB_Memory"."Clock_1Hz"))
	    OR (#ix_ChuteJam OR #sx_ChuteJam) AND "DB_Memory"."Clock_2Hz";

	    //Send RTR signal to the sorter
	    #iqUDT_HandShakeUp.RTR := #ix_SafetyOk AND NOT (#ix_ChuteJam OR #sx_ChuteFull)
	    AND NOT #iqUDT_ChuteCommand.DisableFromHMI
	    AND NOT #iqUDT_ChuteCommand.DisableFromHLC;

	END_REGION

	REGION 7 - Statistics

	    // Chute disable from HMI.
	    IF #sUDT_HMIStatus.Specific.DisableFromHMI
	        OR #iqUDT_EquipmentControl.Command.ResetData
	    THEN
	        "FC_Statistics"(ix_Reset := #iqUDT_EquipmentControl.Command.ResetData,
	                        ix_Activate := #sUDT_HMIStatus.Specific.DisableFromHMI,
	                        ix_RTrigActivate := #sR_TRIG_DisableFromHMI.Q,
	                        iqUDT_Statistics := #iqUDT_Statistics.DisableFromHMI);
	    END_IF;

	    // Chute disable from HLC
	    IF #sUDT_HMIStatus.Specific.DisableFromHLC
	        OR #iqUDT_EquipmentControl.Command.ResetData
	    THEN
	        "FC_Statistics"(ix_Reset := #iqUDT_EquipmentControl.Command.ResetData,
	                        ix_Activate := #sUDT_HMIStatus.Specific.DisableFromHLC,
	                        ix_RTrigActivate := #sR_TRIG_DisableFromHLC.Q,
	                        iqUDT_Statistics := #iqUDT_Statistics.DisableFromHLC);
	    END_IF;

	    //Chute full
	    IF #sUDT_HMIStatus.Specific.ChuteFull
	        OR #iqUDT_EquipmentControl.Command.ResetData
	    THEN

	        "FC_Statistics"(ix_Reset := #iqUDT_EquipmentControl.Command.ResetData,
	                        ix_Activate := #sUDT_HMIStatus.Specific.ChuteFull,
	                        ix_RTrigActivate := #sR_TRIG_ChuteFull.Q,
	                        iqUDT_Statistics := #iqUDT_Statistics.ChuteFull);

	    END_IF;

	    //Chute half full
	    IF #sUDT_HMIStatus.Specific.ChuteHalfFull
	        OR #iqUDT_EquipmentControl.Command.ResetData
	    THEN

	        "FC_Statistics"(ix_Reset := #iqUDT_EquipmentControl.Command.ResetData,
	                        ix_Activate := #sUDT_HMIStatus.Specific.ChuteHalfFull,
	                        ix_RTrigActivate := #sR_TRIG_ChuteHalfFull.Q,
	                        iqUDT_Statistics := #iqUDT_Statistics.ChuteHalfFull);

	    END_IF;

	    //Chute jam
	    IF #sUDT_HMIStatus.Specific.ChuteJam
	        OR #iqUDT_EquipmentControl.Command.ResetData
	    THEN

	        "FC_Statistics"(ix_Reset := #iqUDT_EquipmentControl.Command.ResetData,
	                        ix_Activate := #sUDT_HMIStatus.Specific.ChuteJam,
	                        ix_RTrigActivate := #sR_TRIG_ChuteJam.Q,
	                        iqUDT_Statistics := #iqUDT_Statistics.ChuteJam);

	    END_IF;

	END_REGION

	REGION 8 - Status

	    //Error active
	    #sUDT_CommonStatus.Error := NOT #ix_HardwareOk OR NOT #ix_SafetyOk OR #sx_ChuteJam;

	    //Automation ON
	    #sUDT_CommonStatus.AutoON := #iqUDT_EquipmentControl.Command.AutomaticOn;

	    // Energy save active
	    #sUDT_CommonStatus.EnergySave := #ix_EnergySave;

	    // Running
	    #sUDT_CommonStatus.Running := #sUDT_CommonStatus.AutoON AND NOT #sUDT_CommonStatus.Error;

	    // Stopped
	    #sUDT_CommonStatus.Stopped := NOT #sUDT_CommonStatus.AutoON OR #sUDT_CommonStatus.Error;

	    // Safety not ok
	    #sUDT_CommonStatus.SafetyStop := NOT #ix_SafetyOk;

	    // Chute disabled
	    IF #sUDT_HMIStatus.Specific.DisableFromHMI OR #sUDT_HMIStatus.Specific.DisableFromHLC AND NOT #sUDT_CommonStatus.SafetyStop
	    THEN
	        #sUDT_HMIStatus.Status := "DB_HMIStatusConfiguration".DisableByManagement;
	    END_IF;

	    // Chute Half Full
	    IF #sUDT_HMIStatus.Specific.ChuteHalfFull AND NOT #sUDT_CommonStatus.SafetyStop
	    THEN
	        #sUDT_HMIStatus.Status := "DB_HMIStatusConfiguration".ChuteHalfFull;
	    END_IF;

	    //Chute Full
	    IF #sUDT_HMIStatus.Specific.ChuteFull AND NOT #sUDT_CommonStatus.SafetyStop
	    THEN
	        #sUDT_HMIStatus.Status := "DB_HMIStatusConfiguration".ChuteFull;
	    END_IF;

	    //Chute Jam
	    IF #sUDT_HMIStatus.Specific.ChuteJam AND NOT #sUDT_CommonStatus.SafetyStop
	    THEN
	        #sUDT_HMIStatus.Status := "DB_HMIStatusConfiguration".PECJam;
	    END_IF;

	    //Collecting F_TRIG on chute full, half full, jam or chute disabled status to update common status
	    #sF_TRIG_UpdateStatus(CLK := #sUDT_HMIStatus.Specific.ChuteHalfFull OR #sUDT_HMIStatus.Specific.ChuteFull
	                          OR #sUDT_HMIStatus.Specific.ChuteJam OR #sUDT_HMIStatus.Specific.DisableFromHMI
	                          OR #sUDT_HMIStatus.Specific.DisableFromHLC);

	    // HMI status update
	    IF #sUDT_CommonStatusOld <> #sUDT_CommonStatus OR #sF_TRIG_UpdateStatus.Q  // update on change
	    THEN
	        // HMI status initialization
	        #sUDT_HMIStatus.Status := 0;

	        // Energy save
	        IF #sUDT_CommonStatus.EnergySave
	        THEN
	            #sUDT_HMIStatus.Status := "DB_HMIStatusConfiguration".EnergySave;
	        END_IF;

	        // Running
	        IF #sUDT_CommonStatus.Running
	        THEN
	            #sUDT_HMIStatus.Status := "DB_HMIStatusConfiguration".Running;
	        END_IF;

	        // Stopped
	        IF #sUDT_CommonStatus.Stopped
	        THEN
	            #sUDT_HMIStatus.Status := "DB_HMIStatusConfiguration".Stopped;
	        END_IF;

	        // Error
	        IF #sUDT_CommonStatus.Error
	        THEN
	            #sUDT_HMIStatus.Status := "DB_HMIStatusConfiguration".Stopped;
	        END_IF;

	        // Safety stop
	        IF #sUDT_CommonStatus.SafetyStop
	        THEN
	            #sUDT_HMIStatus.Status := "DB_HMIStatusConfiguration".SafetyStop;
	        END_IF;

	        #sUDT_CommonStatusOld := #sUDT_CommonStatus;              // Copy status to memory
	        #qUDT_Status := #sUDT_CommonStatus;                       // Copy status to output

	    END_IF;

	    // Copy HMI status to output
	    #qUDT_HMIStatus := #sUDT_HMIStatus;

	END_REGION

	REGION 9 - Report to control block

	    // Function to manage report between control block and conveyor block
	    "FC_EquipmentReport"(iUDT_Status := #sUDT_CommonStatus,
	                         iqUDT_Control := #iqUDT_EquipmentControl);

	END_REGION

	REGION 10 - Equipment staus message

	    IF NOT #iqUDT_EquipmentControl.Command.AutomaticOn
	    THEN
	        #ss_StatusCode := '006'; //Inactive
	    ELSIF #sx_ChuteJam
	    THEN
	        #ss_StatusCode := '002';  //Chute Jam
	    ELSIF #sx_ChuteFull
	    THEN
	        #ss_StatusCode := '003';  // Chute Full
	    ELSIF #sx_ChuateHalfFull
	    THEN
	        #ss_StatusCode := '004';  // Chute Half full
	    ELSIF #iqUDT_ChuteCommand.DisableFromHMI OR #iqUDT_ChuteCommand.DisableFromHLC
	    THEN
	        #ss_StatusCode := '005'; // Chute Disabled
	    ELSE
	        #ss_StatusCode := '001'; //Chute is Clear
	    END_IF;

	    #sFB_FedExEquipmentStatusMessage(iUDT_Facility := #iUDT_Facility,
	                                     is_LOConEquipment := #iUDT_ChuteConfiguration.LOConEquipment, // Sorter number
	                                     is_DEPCOD := #iUDT_ChuteConfiguration.DEPCOD,
	                                     is_TYPofEquipment := 'PLC',
	                                     is_NumberOfTheEquipment := #iUDT_ChuteConfiguration.NumberOfTheEquipment,// PLC number
	                                     is_DeviceType := 'CHUTES',
	                                     is_DeviceID := #iUDT_ChuteConfiguration."Device ID", //Chute number
	                                     is_StatusCode := #ss_StatusCode,
	                                     qx_Error => #sx_MessageError,
	                                     iqUDT_FifoHeader := #iqUDT_FifoHighPriorityHLC,
	                                     iqa_FifoData := #iqa_FifoHighPriorityHLC);

	END_REGION

	REGION 11 XBS interface
	    // Map chute status to sorter
	    #qUDT_StatusToXBS.Full := #sUDT_HMIStatus.Specific.ChuteFull;
	    #qUDT_StatusToXBS.HalfFull := #sUDT_HMIStatus.Specific.ChuteHalfFull;
	    #qUDT_StatusToXBS.ReadyToReceive := NOT #sUDT_CommonStatus.Error AND #sUDT_CommonStatus.AutoON;
	    #qUDT_StatusToXBS.Running := #sUDT_CommonStatus.Running;
	    #qUDT_StatusToXBS.Fault := #sUDT_CommonStatus.Error;
	    #qUDT_StatusToXBS.Warning := #sUDT_CommonStatus.Warning;
	END_REGION

END_FUNCTION_BLOCK

FUNCTION_BLOCK "FB_FedExPolisorterGlobalEquipmentStatus"
{ S7_Optimized_Access := 'TRUE' }
VERSION : 0.1
// ATTRIBUTES
// AUTO_NUMBER = True
// BLOCK_NUMBER = 81
// END_ATTRIBUTES
   VAR_INPUT
      iUDT_FedExFacility { ExternalAccessible := 'False'; ExternalVisible := 'False'; ExternalWritable := 'False'} : "UDT_FedExFacility";   // System configuration
      is_LOConEquipment { ExternalAccessible := 'False'; ExternalVisible := 'False'; ExternalWritable := 'False'} : String[3];   // Location of the equipment
      is_DEPCOD { ExternalAccessible := 'False'; ExternalVisible := 'False'; ExternalWritable := 'False'} : String[6];   // Depot Code
      is_TYPofEquipment { ExternalAccessible := 'False'; ExternalVisible := 'False'; ExternalWritable := 'False'} : String[3];   // Type of equipment
      is_NumberOfTheEquipment { ExternalAccessible := 'False'; ExternalVisible := 'False'; ExternalWritable := 'False'} : String[3];   // Number of the equipment 001-999
      ix_Chute1Jam { ExternalAccessible := 'False'; ExternalVisible := 'False'; ExternalWritable := 'False'} : Bool;   // Chute 1 jam error
      is_Chute1Name { ExternalAccessible := 'False'; ExternalVisible := 'False'; ExternalWritable := 'False'} : String[6];   // Chute 1 physical name
      iUDT_Chute1Status { ExternalAccessible := 'False'; ExternalVisible := 'False'; ExternalWritable := 'False'} : "UDT_CommonStatus";
      ix_Chute2Jam { ExternalAccessible := 'False'; ExternalVisible := 'False'; ExternalWritable := 'False'} : Bool;   // Chute 2 jam error
      is_Chute2Name { ExternalAccessible := 'False'; ExternalVisible := 'False'; ExternalWritable := 'False'} : String[6];   // Chute 2 physical name
      i_UDT_Chute2Status { ExternalAccessible := 'False'; ExternalVisible := 'False'; ExternalWritable := 'False'} : "UDT_CommonStatus";
      ix_Chute3Jam { ExternalAccessible := 'False'; ExternalVisible := 'False'; ExternalWritable := 'False'} : Bool;   // Chute 3 jam error
      is_Chute3Name { ExternalAccessible := 'False'; ExternalVisible := 'False'; ExternalWritable := 'False'} : String[6];   // Chute 3 physical name
      iUDT_Chute3Status { ExternalAccessible := 'False'; ExternalVisible := 'False'; ExternalWritable := 'False'} : "UDT_CommonStatus";
      ix_Chute4Jam { ExternalAccessible := 'False'; ExternalVisible := 'False'; ExternalWritable := 'False'} : Bool;   // Chute 4 jam error
      is_Chute4Name { ExternalAccessible := 'False'; ExternalVisible := 'False'; ExternalWritable := 'False'} : String[6];   // Chute 4 physical name
      iUDT_Chute4Status { ExternalAccessible := 'False'; ExternalVisible := 'False'; ExternalWritable := 'False'} : "UDT_CommonStatus";
      ix_Chute5Jam { ExternalAccessible := 'False'; ExternalVisible := 'False'; ExternalWritable := 'False'} : Bool;   // Chute 5 jam error
      is_Chute5Name { ExternalAccessible := 'False'; ExternalVisible := 'False'; ExternalWritable := 'False'} : String[6];   // Chute 5 physical name
      iUDT_Chute5Status { ExternalAccessible := 'False'; ExternalVisible := 'False'; ExternalWritable := 'False'} : "UDT_CommonStatus";
      ix_Chute6Jam { ExternalAccessible := 'False'; ExternalVisible := 'False'; ExternalWritable := 'False'} : Bool;   // Chute 6 jam error
      is_Chute6Name { ExternalAccessible := 'False'; ExternalVisible := 'False'; ExternalWritable := 'False'} : String[6];   // Chute 6 physical name
      iUDT_Chute6Status { ExternalAccessible := 'False'; ExternalVisible := 'False'; ExternalWritable := 'False'} : "UDT_CommonStatus";
      ix_Chute7Jam { ExternalAccessible := 'False'; ExternalVisible := 'False'; ExternalWritable := 'False'} : Bool;
      is_Chute7Name { ExternalAccessible := 'False'; ExternalVisible := 'False'; ExternalWritable := 'False'} : String[6];
      iUDT_Chute7Status { ExternalAccessible := 'False'; ExternalVisible := 'False'; ExternalWritable := 'False'} : "UDT_CommonStatus";
      ix_Chute8Jam { ExternalAccessible := 'False'; ExternalVisible := 'False'; ExternalWritable := 'False'} : Bool;
      is_Chute8Name { ExternalAccessible := 'False'; ExternalVisible := 'False'; ExternalWritable := 'False'} : String[6];
      iUDT_Chute8Status { ExternalAccessible := 'False'; ExternalVisible := 'False'; ExternalWritable := 'False'} : "UDT_CommonStatus";
      ix_Chute9Jam { ExternalAccessible := 'False'; ExternalVisible := 'False'; ExternalWritable := 'False'} : Bool;
      is_Chute9Name { ExternalAccessible := 'False'; ExternalVisible := 'False'; ExternalWritable := 'False'} : String[6];
      iUDT_Chute9Status { ExternalAccessible := 'False'; ExternalVisible := 'False'; ExternalWritable := 'False'} : "UDT_CommonStatus";
      ix_Chute10Jam { ExternalAccessible := 'False'; ExternalVisible := 'False'; ExternalWritable := 'False'} : Bool;
      is_Chute10Name { ExternalAccessible := 'False'; ExternalVisible := 'False'; ExternalWritable := 'False'} : String[6];
      iUDT_Chute10Status { ExternalAccessible := 'False'; ExternalVisible := 'False'; ExternalWritable := 'False'} : "UDT_CommonStatus";
      ix_Polisorter1Jam { ExternalAccessible := 'False'; ExternalVisible := 'False'; ExternalWritable := 'False'} : Bool;   // Polisorter 1 jam error
      ix_Polisorter2Jam { ExternalAccessible := 'False'; ExternalVisible := 'False'; ExternalWritable := 'False'} : Bool;   // Polisorter 2 jam error
      ix_Polisorter3Jam { ExternalAccessible := 'False'; ExternalVisible := 'False'; ExternalWritable := 'False'} : Bool;   // Polisorter 3 jam error
      ix_Polisorter4Jam { ExternalAccessible := 'False'; ExternalVisible := 'False'; ExternalWritable := 'False'} : Bool;   // Polisorter 4 jam error
      iUDT_Polisorter1CommonStatus { ExternalAccessible := 'False'; ExternalVisible := 'False'; ExternalWritable := 'False'} : "UDT_CommonStatus";   // Polisorter 1 common status
      iUDT_Polisorter2CommonStatus { ExternalAccessible := 'False'; ExternalVisible := 'False'; ExternalWritable := 'False'} : "UDT_CommonStatus";   // Polisorter 2 common status
      iUDT_Polisorter3CommonStatus { ExternalAccessible := 'False'; ExternalVisible := 'False'; ExternalWritable := 'False'} : "UDT_CommonStatus";   // Polisorter 3 common status
      iUDT_Polisorter4CommonStatus { ExternalAccessible := 'False'; ExternalVisible := 'False'; ExternalWritable := 'False'} : "UDT_CommonStatus";   // Polisorter 4 common status
   END_VAR

   VAR_IN_OUT
      iUDT_FedExCommands : "UDT_FedExCommands";   // Commands sent by uDS
      iqUDT_FifoHeader : "UDT_FifoHeader";   // Fifo header
      iqa_FifoData : Array[*] of "UDT_Message";   // Fifo data
   END_VAR

   VAR
      sFB_FedExEquipmentStatusMessageChutes { ExternalAccessible := 'False'; ExternalVisible := 'False'; ExternalWritable := 'False'; S7_SetPoint := 'False'} : "FB_FedExEquipmentStatusMessage";   // Equipment status message for chutes
      sFB_FedExEquipmentStatusMessageSorter { ExternalAccessible := 'False'; ExternalVisible := 'False'; ExternalWritable := 'False'; S7_SetPoint := 'False'} : "FB_FedExEquipmentStatusMessage";   // Equipment status message for sorter
      sa_ChuteStatus { ExternalAccessible := 'False'; ExternalVisible := 'False'; ExternalWritable := 'False'} : Array[1..10] of String[3];   // Chute status array
      sa_ChuteStatus_OLD { ExternalAccessible := 'False'; ExternalVisible := 'False'; ExternalWritable := 'False'} : Array[1..10] of String[3];   // ChuteStatusOLD
      sa_ChuteName { ExternalAccessible := 'False'; ExternalVisible := 'False'; ExternalWritable := 'False'} : Array[1..10] of String[6];   // Chute name array
      ss_SorterStatus { ExternalAccessible := 'False'; ExternalVisible := 'False'; ExternalWritable := 'False'} : String[3];   // Sorter status
      ss_SorterStatus_OLD { ExternalAccessible := 'False'; ExternalVisible := 'False'; ExternalWritable := 'False'} : String[3];   // Sorter status OLD
      sR_TRIG_SorterEstop {InstructionName := 'R_TRIG'; LibVersion := '1.0'; ExternalAccessible := 'False'; ExternalVisible := 'False'; ExternalWritable := 'False'; S7_SetPoint := 'False'} : R_TRIG;   // Sorter Estop R_TRIG
      sR_TRIG_SorterJam {InstructionName := 'R_TRIG'; LibVersion := '1.0'; ExternalAccessible := 'False'; ExternalVisible := 'False'; ExternalWritable := 'False'; S7_SetPoint := 'False'} : R_TRIG;   // Sorter Jam R_TRIG
      sR_TRIG_SorterStopped {InstructionName := 'R_TRIG'; LibVersion := '1.0'; ExternalAccessible := 'False'; ExternalVisible := 'False'; ExternalWritable := 'False'; S7_SetPoint := 'False'} : R_TRIG;   // Sorter stop R_TRIG
      sR_TRIG_SorterRunning {InstructionName := 'R_TRIG'; LibVersion := '1.0'; ExternalAccessible := 'False'; ExternalVisible := 'False'; ExternalWritable := 'False'; S7_SetPoint := 'False'} : R_TRIG;   // Sorter running R_TRIG
      sFB_TimerOnOffDelay_FullChute1 { ExternalAccessible := 'False'; ExternalVisible := 'False'; ExternalWritable := 'False'; S7_SetPoint := 'False'} : "FB_TimerOnOffDelay";
      sFB_TimerOnOffDelay_FullChute2 { ExternalAccessible := 'False'; ExternalVisible := 'False'; ExternalWritable := 'False'; S7_SetPoint := 'False'} : "FB_TimerOnOffDelay";
      sFB_TimerOnOffDelay_FullChute3 { ExternalAccessible := 'False'; ExternalVisible := 'False'; ExternalWritable := 'False'; S7_SetPoint := 'False'} : "FB_TimerOnOffDelay";
      sFB_TimerOnOffDelay_FullChute4 { ExternalAccessible := 'False'; ExternalVisible := 'False'; ExternalWritable := 'False'; S7_SetPoint := 'False'} : "FB_TimerOnOffDelay";
      sFB_TimerOnOffDelay_FullChute5 { ExternalAccessible := 'False'; ExternalVisible := 'False'; ExternalWritable := 'False'; S7_SetPoint := 'False'} : "FB_TimerOnOffDelay";
      sFB_TimerOnOffDelay_FullChute6 { ExternalAccessible := 'False'; ExternalVisible := 'False'; ExternalWritable := 'False'; S7_SetPoint := 'False'} : "FB_TimerOnOffDelay";
      sFB_TimerOnOffDelay_FullChute7 { ExternalAccessible := 'False'; ExternalVisible := 'False'; ExternalWritable := 'False'; S7_SetPoint := 'False'} : "FB_TimerOnOffDelay";
      sFB_TimerOnOffDelay_FullChute8 { ExternalAccessible := 'False'; ExternalVisible := 'False'; ExternalWritable := 'False'; S7_SetPoint := 'False'} : "FB_TimerOnOffDelay";
      sFB_TimerOnOffDelay_FullChute9 { ExternalAccessible := 'False'; ExternalVisible := 'False'; ExternalWritable := 'False'; S7_SetPoint := 'False'} : "FB_TimerOnOffDelay";
      sFB_TimerOnOffDelay_FullChute10 { ExternalAccessible := 'False'; ExternalVisible := 'False'; ExternalWritable := 'False'; S7_SetPoint := 'False'} : "FB_TimerOnOffDelay";
   END_VAR

   VAR_TEMP
      ti_i : Int;
   END_VAR

   VAR CONSTANT
      ChuteFullDelay : UDInt := 2000;
   END_VAR


BEGIN
	(*
	----------------------------------------------------------------------------------------

	Version history:
	Date        | Version   | Author        | Remark
	----------------------------------------------------------------------------------------
	26/04/2022  | 1.0       | K. Pokorski   | first release MHS TIA 16.0
	21/02/2023  | 4.0       | F.Baten       | 4.0 Release TIA 17.5
	*)

	REGION 1 - Copy chutes name

	    #sa_ChuteName[1] := #is_Chute1Name;
	    #sa_ChuteName[2] := #is_Chute2Name;
	    #sa_ChuteName[3] := #is_Chute3Name;
	    #sa_ChuteName[4] := #is_Chute4Name;
	    #sa_ChuteName[5] := #is_Chute5Name;
	    #sa_ChuteName[6] := #is_Chute6Name;
	    #sa_ChuteName[7] := #is_Chute7Name;
	    #sa_ChuteName[8] := #is_Chute8Name;
	    #sa_ChuteName[9] := #is_Chute9Name;
	    #sa_ChuteName[10] := #is_Chute10Name;

	END_REGION

	REGION 2 - Creating chute status

	    #sFB_TimerOnOffDelay_FullChute1(iudi_OnDelayTime := #ChuteFullDelay,
	                                    ix_SignalToDelay := #iUDT_Chute1Status.Dieback OR #iUDT_Chute1Status.Halted);


	    IF #ix_Chute1Jam THEN
	        #sa_ChuteStatus[1] := '002';
	    ELSIF #sFB_TimerOnOffDelay_FullChute1.qx_DelayedSignal THEN
	        #sa_ChuteStatus[1] := '003';
	        // ELSIF NOT #i_UDT_Chute1Status.AutoON THEN
	        //     #sa_ChuteStatus[1] := '006';
	    ELSE
	        #sa_ChuteStatus[1] := '001';
	    END_IF;

	    #sFB_TimerOnOffDelay_FullChute2(iudi_OnDelayTime := #ChuteFullDelay,
	                                    ix_SignalToDelay := #i_UDT_Chute2Status.Dieback OR #i_UDT_Chute2Status.Halted);

	    IF #ix_Chute2Jam THEN
	        #sa_ChuteStatus[2] := '002';
	    ELSIF #sFB_TimerOnOffDelay_FullChute2.qx_DelayedSignal THEN
	        #sa_ChuteStatus[2] := '003';
	        // ELSIF NOT #i_UDT_Chute2Status.AutoON THEN
	        //     #sa_ChuteStatus[2] := '006';
	    ELSE
	        #sa_ChuteStatus[2] := '001';
	    END_IF;

	    #sFB_TimerOnOffDelay_FullChute3(iudi_OnDelayTime := #ChuteFullDelay,
	                                    ix_SignalToDelay := #iUDT_Chute3Status.Dieback OR #iUDT_Chute3Status.Halted);

	    IF #ix_Chute3Jam THEN
	        #sa_ChuteStatus[3] := '002';
	    ELSIF #sFB_TimerOnOffDelay_FullChute3.qx_DelayedSignal THEN
	        #sa_ChuteStatus[3] := '003';
	        // ELSIF NOT #i_UDT_Chute3Status.AutoON THEN
	        //     #sa_ChuteStatus[3] := '006';
	    ELSE
	        #sa_ChuteStatus[3] := '001';
	    END_IF;

	    #sFB_TimerOnOffDelay_FullChute4(iudi_OnDelayTime := #ChuteFullDelay,
	                                    ix_SignalToDelay := #iUDT_Chute4Status.Dieback OR #iUDT_Chute4Status.Halted);

	    IF #ix_Chute4Jam THEN
	        #sa_ChuteStatus[4] := '002';
	    ELSIF #sFB_TimerOnOffDelay_FullChute4.qx_DelayedSignal THEN
	        #sa_ChuteStatus[4] := '003';
	        // ELSIF NOT #i_UDT_Chute4Status.AutoON THEN
	        //     #sa_ChuteStatus[4] := '006';
	    ELSE
	        #sa_ChuteStatus[4] := '001';
	    END_IF;

	    #sFB_TimerOnOffDelay_FullChute5(iudi_OnDelayTime := #ChuteFullDelay,
	                                    ix_SignalToDelay := #iUDT_Chute5Status.Dieback OR #iUDT_Chute5Status.Halted);

	    IF #ix_Chute5Jam THEN
	        #sa_ChuteStatus[5] := '002';
	    ELSIF #sFB_TimerOnOffDelay_FullChute5.qx_DelayedSignal THEN
	        #sa_ChuteStatus[5] := '003';
	        // ELSIF NOT #i_UDT_Chute5Status.AutoON THEN
	        //     #sa_ChuteStatus[5] := '006';
	    ELSE
	        #sa_ChuteStatus[5] := '001';
	    END_IF;

	    #sFB_TimerOnOffDelay_FullChute6(iudi_OnDelayTime := #ChuteFullDelay,
	                                    ix_SignalToDelay := #iUDT_Chute6Status.Dieback OR #iUDT_Chute6Status.Halted);

	    IF #ix_Chute6Jam THEN
	        #sa_ChuteStatus[6] := '002';
	    ELSIF #sFB_TimerOnOffDelay_FullChute6.qx_DelayedSignal THEN
	        #sa_ChuteStatus[6] := '003';
	        // ELSIF NOT #i_UDT_Chute6Status.AutoON THEN
	        //     #sa_ChuteStatus[6] := '006';
	    ELSE
	        #sa_ChuteStatus[6] := '001';
	    END_IF;


	    #sFB_TimerOnOffDelay_FullChute7(iudi_OnDelayTime := #ChuteFullDelay,
	                                    ix_SignalToDelay := #iUDT_Chute7Status.Dieback OR #iUDT_Chute7Status.Halted);


	    IF #ix_Chute7Jam THEN
	        #sa_ChuteStatus[7] := '002';
	    ELSIF #sFB_TimerOnOffDelay_FullChute7.qx_DelayedSignal THEN
	        #sa_ChuteStatus[7] := '003';
	        // ELSIF NOT #i_UDT_Chute7Status.AutoON THEN
	        //     #sa_ChuteStatus[7] := '006';
	    ELSE
	        #sa_ChuteStatus[7] := '001';
	    END_IF;

	    #sFB_TimerOnOffDelay_FullChute8(iudi_OnDelayTime := #ChuteFullDelay,
	                                    ix_SignalToDelay := #iUDT_Chute8Status.Dieback OR #iUDT_Chute8Status.Halted);

	    IF #ix_Chute8Jam THEN
	        #sa_ChuteStatus[8] := '002';
	    ELSIF #sFB_TimerOnOffDelay_FullChute8.qx_DelayedSignal THEN
	        #sa_ChuteStatus[8] := '003';
	        // ELSIF NOT #i_UDT_Chute8Status.AutoON THEN
	        //     #sa_ChuteStatus[8] := '006';
	    ELSE
	        #sa_ChuteStatus[8] := '001';
	    END_IF;

	    #sFB_TimerOnOffDelay_FullChute9(iudi_OnDelayTime := #ChuteFullDelay,
	                                    ix_SignalToDelay := #iUDT_Chute9Status.Dieback OR #iUDT_Chute9Status.Halted);

	    IF #ix_Chute9Jam THEN
	        #sa_ChuteStatus[9] := '002';
	    ELSIF #sFB_TimerOnOffDelay_FullChute9.qx_DelayedSignal THEN
	        #sa_ChuteStatus[9] := '003';
	        // ELSIF NOT #i_UDT_Chute9Status.AutoON THEN
	        //     #sa_ChuteStatus[9] := '006';
	    ELSE
	        #sa_ChuteStatus[9] := '001';
	    END_IF;

	    #sFB_TimerOnOffDelay_FullChute10(iudi_OnDelayTime := #ChuteFullDelay,
	                                     ix_SignalToDelay := #iUDT_Chute10Status.Dieback OR #iUDT_Chute10Status.Halted);

	    IF #ix_Chute10Jam THEN
	        #sa_ChuteStatus[10] := '002';
	    ELSIF #sFB_TimerOnOffDelay_FullChute10.qx_DelayedSignal THEN
	        #sa_ChuteStatus[10] := '003';
	        // ELSIF NOT #i_UDT_Chute10Status.AutoON THEN
	        //     #sa_ChuteStatus[10] := '006';
	    ELSE
	        #sa_ChuteStatus[10] := '001';
	    END_IF;

	END_REGION

	REGION 3 - Sending equipment status message for chutes

	    FOR #ti_i := 1 TO 10 DO

	        IF #sa_ChuteStatus_OLD[#ti_i] <> #sa_ChuteStatus[#ti_i]
	            OR #iUDT_FedExCommands.UploadChuteStatus.NewMessage
	            OR #iUDT_FedExCommands.UploadAllStatus.NewMessage
	        THEN

	            #sFB_FedExEquipmentStatusMessageChutes(iUDT_Facility := #iUDT_FedExFacility,
	                                                   is_LOConEquipment := #is_LOConEquipment,
	                                                   is_DEPCOD := #is_DEPCOD,
	                                                   is_TYPofEquipment := #is_TYPofEquipment,
	                                                   is_NumberOfTheEquipment := #is_NumberOfTheEquipment,
	                                                   is_DeviceType := 'CHUTES',
	                                                   is_DeviceID := #sa_ChuteName[#ti_i],
	                                                   is_StatusCode := #sa_ChuteStatus[#ti_i],
	                                                   iqUDT_FifoHeader := #iqUDT_FifoHeader,
	                                                   iqa_FifoData := #iqa_FifoData);
	        END_IF;


	    END_FOR;

	END_REGION

	REGION 4 - Detecting triggers in sorter status

	    #sR_TRIG_SorterEstop(CLK := #iUDT_Polisorter1CommonStatus.SafetyStop
	                         OR #iUDT_Polisorter2CommonStatus.SafetyStop
	                         OR #iUDT_Polisorter3CommonStatus.SafetyStop
	                         OR #iUDT_Polisorter4CommonStatus.SafetyStop);

	    #sR_TRIG_SorterJam(CLK := #ix_Polisorter1Jam
	                       OR #ix_Polisorter2Jam
	                       OR #ix_Polisorter3Jam
	                       OR #ix_Polisorter4Jam);

	    #sR_TRIG_SorterStopped(CLK := #iUDT_Polisorter1CommonStatus.Stopped
	                           AND #iUDT_Polisorter2CommonStatus.Stopped
	                           AND #iUDT_Polisorter3CommonStatus.Stopped
	                           AND #iUDT_Polisorter4CommonStatus.Stopped);

	    #sR_TRIG_SorterRunning(CLK := #iUDT_Polisorter1CommonStatus.Running
	                           OR #iUDT_Polisorter2CommonStatus.Running
	                           OR #iUDT_Polisorter3CommonStatus.Running
	                           OR #iUDT_Polisorter4CommonStatus.Running);
	END_REGION


	REGION 5 - Creating sorter status

	    IF #sR_TRIG_SorterEstop.Q
	    THEN
	        #ss_SorterStatus := '004';
	    ELSIF #sR_TRIG_SorterJam.Q
	    THEN
	        #ss_SorterStatus := '003';
	    ELSIF #sR_TRIG_SorterStopped.Q
	    THEN
	        #ss_SorterStatus := '002';
	    ELSIF #sR_TRIG_SorterRunning.Q
	    THEN
	        #ss_SorterStatus := '001';

	    END_IF;
	END_REGION

	REGION 6 - Sending sorter status

	    IF #ss_SorterStatus_OLD <> #ss_SorterStatus
	        OR #iUDT_FedExCommands.UploadAllStatus.NewMessage THEN

	        #sFB_FedExEquipmentStatusMessageSorter(iUDT_Facility := #iUDT_FedExFacility,
	                                               is_LOConEquipment := #is_LOConEquipment,
	                                               is_DEPCOD := #is_DEPCOD,
	                                               is_TYPofEquipment := #is_TYPofEquipment,
	                                               is_NumberOfTheEquipment := #is_NumberOfTheEquipment,
	                                               is_DeviceType := 'PLC001',
	                                               is_DeviceID := '000001',
	                                               is_StatusCode := #ss_SorterStatus,
	                                               iqUDT_FifoHeader := #iqUDT_FifoHeader,
	                                               iqa_FifoData := #iqa_FifoData);

	    END_IF;

	END_REGION

	REGION 7 - Store old statuses

	    #ss_SorterStatus_OLD := #ss_SorterStatus;
	    #sa_ChuteStatus_OLD := #sa_ChuteStatus;

	END_REGION

	REGION 8 - Reset uDS commands

	    #iUDT_FedExCommands.UploadAllStatus.NewMessage := FALSE;
	    #iUDT_FedExCommands.UploadChuteStatus.NewMessage := FALSE;

	END_REGION





END_FUNCTION_BLOCK

FUNCTION_BLOCK "FB_FedExPolisorterSortResult"
{ S7_Optimized_Access := 'TRUE' }
VERSION : 0.1
// ATTRIBUTES
// AUTO_NUMBER = True
// BLOCK_NUMBER = 82
// END_ATTRIBUTES
   VAR_INPUT
      iUDT_PolisorterInterface { ExternalAccessible := 'False'; ExternalVisible := 'False'; ExternalWritable := 'False'} : "UDT_PolisorterInterface";   // Polisorter interface
      ia_PolisorterDestinations { ExternalAccessible := 'False'; ExternalVisible := 'False'; ExternalWritable := 'False'} : Array[1..3] of "UDT_FedExDestinations";   // Polisorter destinations
      is_RejectChute { ExternalAccessible := 'False'; ExternalVisible := 'False'; ExternalWritable := 'False'} : String[6];   // Physical Destination of custom reject chute
      is_NotReachableDestination1 { ExternalAccessible := 'False'; ExternalVisible := 'False'; ExternalWritable := 'False'} : String[6];
      is_NotReachableDestination2 { ExternalAccessible := 'False'; ExternalVisible := 'False'; ExternalWritable := 'False'} : String[6];
      ii_DVMessageSendPoint { ExternalAccessible := 'False'; ExternalVisible := 'False'; ExternalWritable := 'False'} : Int;   // DV message send point
      ix_FinalSorter { ExternalAccessible := 'False'; ExternalVisible := 'False'; ExternalWritable := 'False'} : Bool;   // True when sorter is last sorter in the system
   END_VAR

   VAR_IN_OUT
      iqi_GINDVMessage { ExternalAccessible := 'False'; ExternalVisible := 'False'; ExternalWritable := 'False'} : Int;   // GIN number
   END_VAR

   VAR
      sF_TRIG_Newparcel {InstructionName := 'F_TRIG'; LibVersion := '1.0'; ExternalAccessible := 'False'; ExternalVisible := 'False'; ExternalWritable := 'False'; S7_SetPoint := 'False'} : F_TRIG;   // New parcel detected at the end of Polisorter
      sdw_ReasonCode { ExternalAccessible := 'False'; ExternalVisible := 'False'; ExternalWritable := 'False'} : DWord;
      si_LastGin { ExternalAccessible := 'False'; ExternalVisible := 'False'; ExternalWritable := 'False'} : Int;   // GIN number from previous cycle
      si_GINDVMessage { ExternalAccessible := 'False'; ExternalVisible := 'False'; ExternalWritable := 'False'} : Int;   // GIN number
      si_StringLen { ExternalAccessible := 'False'; ExternalVisible := 'False'; ExternalWritable := 'False'} : Int;   // Length of actual destination
      si_LenFillLoop { ExternalAccessible := 'False'; ExternalVisible := 'False'; ExternalWritable := 'False'} : Int;
      sx_SendToNextScan { ExternalAccessible := 'False'; ExternalVisible := 'False'; ExternalWritable := 'False'} : Bool;
      sx_EndOfTracking { ExternalAccessible := 'False'; ExternalVisible := 'False'; ExternalWritable := 'False'} : Bool;
      sx_UnknownReason { ExternalAccessible := 'False'; ExternalVisible := 'False'; ExternalWritable := 'False'} : Bool;
   END_VAR

   VAR_TEMP
      ti_LC_Positions : Int;   // Loop counter
      ti_LC_LenFillLoop : Int;   // Loop counter
      ti_LC_Destinations : Int;   // Loop counter
      tw_HTA_RET_VAL : Word;
   END_VAR


BEGIN
	(*
	----------------------------------------------------------------------------------------

	Version history:
	Date        | Version   | Author        | Remark
	----------------------------------------------------------------------------------------
	26/04/2022  | 1.0       | K. Pokorski   | first release MHS TIA 16.0
	21/02/2023  | 4.0       | F.Baten       | 4.0 Release TIA 17.5

	*)
	REGION 1 - Creating sort reason code

	    #sF_TRIG_Newparcel(CLK := #ii_DVMessageSendPoint <> 0);

	    IF #sF_TRIG_Newparcel.Q AND (#si_LastGin) > 0 AND (#si_LastGin <= 9999) THEN
	        #sx_EndOfTracking := FALSE;
	        #sx_UnknownReason := FALSE;

	        IF #ix_FinalSorter THEN
	            #sx_SendToNextScan := TRUE;
	        ELSE
	            #sx_SendToNextScan := FALSE;
	        END_IF;

	        #si_GINDVMessage := #si_LastGin;
	        // No destination received at all
	        IF STRING_TO_DINT("DB_GIN".GIN[#si_GINDVMessage].FedEx.Destination1) = 0 THEN
	            IF "DB_GIN".GIN[#si_GINDVMessage].FedEx.CustomerID <> 0 THEN
	                "DB_GIN".GIN[#si_GINDVMessage].General.SortStatus.NoDivertCause.NoDestRcv := TRUE;
	                #sx_EndOfTracking := TRUE;
	                // No parcel inducted/Unknown state
	            ELSE
	                #sx_UnknownReason := TRUE;
	            END_IF;

	            FOR #ti_LC_Positions := 1 TO 3 BY 1 DO
	                IF #iUDT_PolisorterInterface.PositionActual = #ti_LC_Positions
	                    OR (#iUDT_PolisorterInterface.PositionActual = 0 AND #iUDT_PolisorterInterface.Positioning AND #iUDT_PolisorterInterface.PositionSetpoint = #ti_LC_Positions)
	                THEN

	                    VAL_STRG(IN := #ia_PolisorterDestinations[#ti_LC_Positions].PhysicalDestination,
	                             SIZE := 6,
	                             PREC := 0,
	                             FORMAT := 0,
	                             P := 1,
	                             OUT => "DB_GIN".GIN[#si_GINDVMessage].FedEx.ActualDestination);

	                    #si_StringLen := LEN("DB_GIN".GIN[#si_GINDVMessage].FedEx.ActualDestination);

	                    IF (#si_StringLen < 6)
	                    THEN
	                        FOR #ti_LC_LenFillLoop := 1 TO 6 - #si_StringLen DO
	                            "DB_GIN".GIN[#si_GINDVMessage].FedEx.ActualDestination := CONCAT(IN1 := '0',
	                                                                                             IN2 := "DB_GIN".GIN[#si_GINDVMessage].FedEx.ActualDestination);
	                            EXIT;

	                        END_FOR;
	                    END_IF;
	                    EXIT;
	                END_IF;
	            END_FOR;



	            "DB_GIN".GIN[#si_GINDVMessage].FedEx.PackageExitPoint := CONCAT(IN1 := 'CHUTE', IN2 := "DB_GIN".GIN[#si_GINDVMessage].FedEx.ActualDestination);
	            "DB_GIN".GIN[#si_GINDVMessage].FedEx.PackageExitState := '1';


	            // Destination received after decision on Polisorter
	        ELSIF STRING_TO_DINT("DB_GIN".GIN[#si_GINDVMessage].FedEx.Destination1) <> 0 AND "DB_GIN".GIN[#si_GINDVMessage].General.SortStatus.NoDivertCause.NoDestRcv
	        THEN
	            "DB_GIN".GIN[#si_GINDVMessage].General.SortStatus.NoDivertCause.DestTooLate := TRUE;
	            "DB_GIN".GIN[#si_GINDVMessage].General.SortStatus.NoDivertCause.NoDestRcv := FALSE;
	            #sx_EndOfTracking := TRUE;



	            FOR #ti_LC_Positions := 1 TO 3 BY 1 DO
	                IF #iUDT_PolisorterInterface.PositionActual = #ti_LC_Positions
	                    OR (#iUDT_PolisorterInterface.PositionActual = 0 AND #iUDT_PolisorterInterface.Positioning AND #iUDT_PolisorterInterface.PositionSetpoint = #ti_LC_Positions)

	                THEN

	                    VAL_STRG(IN := #ia_PolisorterDestinations[#ti_LC_Positions].PhysicalDestination,
	                             SIZE := 6,
	                             PREC := 0,
	                             FORMAT := 0,
	                             P := 1,
	                             OUT => "DB_GIN".GIN[#si_GINDVMessage].FedEx.ActualDestination);

	                    #si_StringLen := LEN("DB_GIN".GIN[#si_GINDVMessage].FedEx.ActualDestination);

	                    IF (#si_StringLen < 6)
	                    THEN
	                        FOR #ti_LC_LenFillLoop := 1 TO 6 - #si_StringLen DO
	                            "DB_GIN".GIN[#si_GINDVMessage].FedEx.ActualDestination := CONCAT(IN1 := '0',
	                                                                                             IN2 := "DB_GIN".GIN[#si_GINDVMessage].FedEx.ActualDestination);
	                            EXIT;

	                        END_FOR;
	                    END_IF;
	                    EXIT;
	                END_IF;
	            END_FOR;




	            "DB_GIN".GIN[#si_GINDVMessage].FedEx.PackageExitPoint := CONCAT(IN1 := 'CHUTE', IN2 := "DB_GIN".GIN[#si_GINDVMessage].FedEx.ActualDestination);
	            "DB_GIN".GIN[#si_GINDVMessage].FedEx.PackageExitState := '1';



	            // Any destination received
	        ELSIF STRING_TO_DINT("DB_GIN".GIN[#si_GINDVMessage].FedEx.Destination1) <> 0 THEN

	            // Destination is not configured
	            IF "DB_GIN".GIN[#si_GINDVMessage].General.SortStatus.NoDivertCause.InvalidDest THEN

	                #sx_EndOfTracking := TRUE;

	                IF "DB_GIN".GIN[#si_GINDVMessage].FedEx.Destination1 = #is_NotReachableDestination1
	                    OR "DB_GIN".GIN[#si_GINDVMessage].FedEx.Destination1 = #is_NotReachableDestination2 THEN

	                    "DB_GIN".GIN[#si_GINDVMessage].General.SortStatus.NoDivertCause.DestNotReachable := TRUE;

	                END_IF;

	                FOR #ti_LC_Positions := 1 TO 3 BY 1 DO
	                    IF #iUDT_PolisorterInterface.PositionActual = #ti_LC_Positions
	                        OR (#iUDT_PolisorterInterface.PositionActual = 0 AND #iUDT_PolisorterInterface.Positioning AND #iUDT_PolisorterInterface.PositionSetpoint = #ti_LC_Positions)

	                    THEN

	                        VAL_STRG(IN := #ia_PolisorterDestinations[#ti_LC_Positions].PhysicalDestination,
	                                 SIZE := 6,
	                                 PREC := 0,
	                                 FORMAT := 0,
	                                 P := 1,
	                                 OUT => "DB_GIN".GIN[#si_GINDVMessage].FedEx.ActualDestination);

	                        #si_StringLen := LEN("DB_GIN".GIN[#si_GINDVMessage].FedEx.ActualDestination);

	                        IF (#si_StringLen < 6)
	                        THEN
	                            FOR #ti_LC_LenFillLoop := 1 TO 6 - #si_StringLen DO
	                                "DB_GIN".GIN[#si_GINDVMessage].FedEx.ActualDestination := CONCAT(IN1 := '0',
	                                                                                                 IN2 := "DB_GIN".GIN[#si_GINDVMessage].FedEx.ActualDestination);
	                                EXIT;

	                            END_FOR;
	                        END_IF;
	                        EXIT;
	                    END_IF;
	                END_FOR;


	                "DB_GIN".GIN[#si_GINDVMessage].FedEx.PackageExitPoint := CONCAT(IN1 := 'CHUTE', IN2 := "DB_GIN".GIN[#si_GINDVMessage].FedEx.ActualDestination);
	                "DB_GIN".GIN[#si_GINDVMessage].FedEx.PackageExitState := '1';


	            ELSE

	                //Destination matching the configuration - searching if Poliosorter is in good position
	                FOR #ti_LC_Positions := 1 TO 3 BY 1 DO
	                    IF #iUDT_PolisorterInterface.PositionActual = #ti_LC_Positions
	                        OR (#iUDT_PolisorterInterface.PositionActual = 0 AND #iUDT_PolisorterInterface.Positioning AND #iUDT_PolisorterInterface.PositionSetpoint = #ti_LC_Positions)

	                    THEN
	                        FOR #ti_LC_Destinations := 0 TO 5 DO
	                            IF (#ia_PolisorterDestinations[#ti_LC_Positions].Destination[#ti_LC_Destinations]) = STRING_TO_DINT("DB_GIN".GIN[#si_GINDVMessage].FedEx.Destination1)

	                            THEN

	                                // Polisorter is in good position
	                                VAL_STRG(IN := #ia_PolisorterDestinations[#ti_LC_Positions].PhysicalDestination,
	                                         SIZE := 6,
	                                         PREC := 0,
	                                         FORMAT := 0,
	                                         P := 1,
	                                         OUT => "DB_GIN".GIN[#si_GINDVMessage].FedEx.ActualDestination);

	                                #si_StringLen := LEN("DB_GIN".GIN[#si_GINDVMessage].FedEx.ActualDestination);

	                                #sx_EndOfTracking := NOT #ix_FinalSorter AND "DB_GIN".GIN[#si_GINDVMessage].FedEx.ActualDestination <> #is_RejectChute;

	                                IF (#si_StringLen < 6)
	                                THEN
	                                    FOR #ti_LC_LenFillLoop := 1 TO 6 - #si_StringLen DO
	                                        "DB_GIN".GIN[#si_GINDVMessage].FedEx.ActualDestination := CONCAT(IN1 := '0',
	                                                                                                         IN2 := "DB_GIN".GIN[#si_GINDVMessage].FedEx.ActualDestination);
	                                        EXIT;

	                                    END_FOR;
	                                END_IF;


	                                EXIT;





	                            END_IF;
	                        END_FOR;
	                        EXIT;
	                    END_IF;
	                END_FOR;

	                // Polisorter in wrong position, Divert failed for some reason
	                IF "DB_GIN".GIN[#si_GINDVMessage].FedEx.ActualDestination = '      ' THEN

	                    "DB_GIN".GIN[#si_GINDVMessage].General.SortStatus.FailedDivert := TRUE;
	                    #sx_EndOfTracking := TRUE;

	                    FOR #ti_LC_Positions := 1 TO 3 BY 1 DO
	                        IF #iUDT_PolisorterInterface.PositionActual = #ti_LC_Positions
	                            OR (#iUDT_PolisorterInterface.PositionActual = 0 AND #iUDT_PolisorterInterface.Positioning AND #iUDT_PolisorterInterface.PositionSetpoint = #ti_LC_Positions)

	                        THEN

	                            VAL_STRG(IN := #ia_PolisorterDestinations[#ti_LC_Positions].PhysicalDestination,
	                                     SIZE := 6,
	                                     PREC := 0,
	                                     FORMAT := 0,
	                                     P := 1,
	                                     OUT => "DB_GIN".GIN[#si_GINDVMessage].FedEx.ActualDestination);

	                            #si_StringLen := LEN("DB_GIN".GIN[#si_GINDVMessage].FedEx.ActualDestination);

	                            IF (#si_StringLen < 6)
	                            THEN
	                                FOR #ti_LC_LenFillLoop := 1 TO 6 - #si_StringLen DO
	                                    "DB_GIN".GIN[#si_GINDVMessage].FedEx.ActualDestination := CONCAT(IN1 := '0',
	                                                                                                     IN2 := "DB_GIN".GIN[#si_GINDVMessage].FedEx.ActualDestination);
	                                    EXIT;

	                                END_FOR;
	                            END_IF;
	                            EXIT;
	                        END_IF;
	                    END_FOR;


	                    "DB_GIN".GIN[#si_GINDVMessage].FedEx.PackageExitPoint := CONCAT(IN1 := 'CHUTE', IN2 := "DB_GIN".GIN[#si_GINDVMessage].FedEx.ActualDestination);
	                    "DB_GIN".GIN[#si_GINDVMessage].FedEx.PackageExitState := '1';

	                    // Polisorter in good position, divert successful
	                ELSE

	                    "DB_GIN".GIN[#si_GINDVMessage].General.SortStatus.GoodDivert := TRUE;
	                    "DB_GIN".GIN[#si_GINDVMessage].FedEx.PackageExitPoint := CONCAT(IN1 := 'CHUTE', IN2 := "DB_GIN".GIN[#si_GINDVMessage].FedEx.ActualDestination);
	                    "DB_GIN".GIN[#si_GINDVMessage].FedEx.PackageExitState := '1';

	                END_IF;


	            END_IF;
	        END_IF;

	        #si_StringLen := LEN("DB_GIN".GIN[#si_GINDVMessage].FedEx.PackageExitPoint);

	        IF (#si_StringLen < 14)
	        THEN
	            FOR #si_LenFillLoop := 1 TO 14 - #si_StringLen DO

	                "DB_GIN".GIN[#si_GINDVMessage].FedEx.PackageExitPoint := CONCAT(IN1 := "DB_GIN".GIN[#si_GINDVMessage].FedEx.PackageExitPoint,
	                                                                                IN2 := ' ');
	            END_FOR;

	        END_IF;

	        #sdw_ReasonCode.%X0 := (#ix_FinalSorter OR (#is_RejectChute = "DB_GIN".GIN[#si_GINDVMessage].FedEx.ActualDestination)) AND ("DB_GIN".GIN[#si_GINDVMessage].General.SortStatus.GoodDivert AND "DB_GIN".GIN[#si_GINDVMessage].FedEx.Destination1 <> '999999');
	        #sdw_ReasonCode.%X1 := "DB_GIN".GIN[#si_GINDVMessage].General.SortStatus.NoDivertCause.InvalidDest AND NOT "DB_GIN".GIN[#si_GINDVMessage].General.SortStatus.NoDivertCause.DestNotReachable;
	        #sdw_ReasonCode.%X2 := "DB_GIN".GIN[#si_GINDVMessage].General.SortStatus.NoDivertCause.NoDestRcv AND NOT #sx_UnknownReason;
	        #sdw_ReasonCode.%X3 := "DB_GIN".GIN[#si_GINDVMessage].General.SortStatus.NoDivertCause.DestTooLate;
	        #sdw_ReasonCode.%X4 := FALSE;
	        #sdw_ReasonCode.%X5 := FALSE;
	        #sdw_ReasonCode.%X6 := FALSE;
	        #sdw_ReasonCode.%X7 := FALSE;
	        #sdw_ReasonCode.%X8 := "DB_GIN".GIN[#si_GINDVMessage].General.SortStatus.FailedDivert;
	        #sdw_ReasonCode.%X9 := FALSE;
	        #sdw_ReasonCode.%X10 := FALSE;
	        #sdw_ReasonCode.%X11 := FALSE;//"DB_GIN".GIN[#si_GIN_DVMessage].General.Lost;
	        #sdw_ReasonCode.%X12 := FALSE;
	        #sdw_ReasonCode.%X13 := FALSE;
	        #sdw_ReasonCode.%X14 := FALSE;
	        #sdw_ReasonCode.%X15 := FALSE;
	        #sdw_ReasonCode.%X16 := #sx_EndOfTracking;
	        #sdw_ReasonCode.%X17 := FALSE;
	        #sdw_ReasonCode.%X18 := FALSE;
	        #sdw_ReasonCode.%X19 := FALSE;
	        #sdw_ReasonCode.%X20 := FALSE;
	        #sdw_ReasonCode.%X21 := FALSE;
	        #sdw_ReasonCode.%X22 := FALSE;
	        #sdw_ReasonCode.%X23 := FALSE;
	        #sdw_ReasonCode.%X24 := FALSE;
	        #sdw_ReasonCode.%X25 := "DB_GIN".GIN[#si_GINDVMessage].General.SortStatus.GoodDivert AND "DB_GIN".GIN[#si_GINDVMessage].FedEx.Destination1 = '999999' AND #ix_FinalSorter;
	        #sdw_ReasonCode.%X26 := (NOT #ix_FinalSorter AND (#is_RejectChute <> "DB_GIN".GIN[#si_GINDVMessage].FedEx.ActualDestination)) AND "DB_GIN".GIN[#si_GINDVMessage].General.SortStatus.GoodDivert;
	        #sdw_ReasonCode.%X27 := FALSE;
	        #sdw_ReasonCode.%X28 := FALSE;
	        #sdw_ReasonCode.%X29 := "DB_GIN".GIN[#si_GINDVMessage].General.SortStatus.NoDivertCause.InvalidDest AND "DB_GIN".GIN[#si_GINDVMessage].General.SortStatus.NoDivertCause.DestNotReachable;
	        #sdw_ReasonCode.%X30 := FALSE;
	        #sdw_ReasonCode.%X31 := #sx_UnknownReason;

	        #tw_HTA_RET_VAL := HTA(IN := #sdw_ReasonCode, N := 4, OUT => "DB_GIN".GIN[#si_GINDVMessage].FedEx.ReasonCode1);


	        #iqi_GINDVMessage := #si_GINDVMessage;


	    END_IF;

	    #si_LastGin := #ii_DVMessageSendPoint;

	END_REGION




END_FUNCTION_BLOCK

FUNCTION_BLOCK "FB_FedExStartOfSort"
TITLE = FB_Heartbeat
{ S7_Optimized_Access := 'TRUE' }
AUTHOR : MHSE
FAMILY : UPS_SpecificCommunication
VERSION : 3.0
// ATTRIBUTES
// AUTO_NUMBER = True
// BLOCK_NUMBER = 83
// END_ATTRIBUTES
//Function block to send and monitor the UPS heartbeat message.
   VAR_INPUT
      ix_StartOfSort { ExternalAccessible := 'False'; ExternalVisible := 'False'; ExternalWritable := 'False'} : Bool;   // Enable Start of sort Message
      ix_EnableSend { ExternalAccessible := 'False'; ExternalVisible := 'False'; ExternalWritable := 'False'} : Bool;   // Enable heartbeat message send
      ix_ResetData { ExternalAccessible := 'False'; ExternalVisible := 'False'; ExternalWritable := 'False'} : Bool;   // Reset statistics
   END_VAR

   VAR_IN_OUT
      iqUDT_FifoHeader : "UDT_FifoHeader";   // FIFO header
      iqs_FifoData : Array[*] of "UDT_Message";   // FIFO data
      iqUDT_Statistics : "UDT_FedExHeartbeatStatistics";   // Statistic strucure
      iqdi_UniqueMsgID { ExternalAccessible := 'False'; ExternalVisible := 'False'; ExternalWritable := 'False'} : DInt;   // Unique message ID integer
   END_VAR

   VAR
      s_R_TRIG_EnableSend {InstructionName := 'R_TRIG'; LibVersion := '1.0'; ExternalAccessible := 'False'; ExternalVisible := 'False'; ExternalWritable := 'False'; S7_SetPoint := 'False'} : R_TRIG;   // Siemens "R_TRIG" - to prepare the rising edge trigger on "ix_EnableSend" signal
      s_R_TRIG_StartOfSort {InstructionName := 'R_TRIG'; LibVersion := '1.0'; ExternalAccessible := 'False'; ExternalVisible := 'False'; ExternalWritable := 'False'; S7_SetPoint := 'False'} : R_TRIG;   // Siemens "R_TRIG" - to prepare the rising edge trigger on "ix_StartOfSort" signal
      s_UDT_MessageArray { ExternalAccessible := 'False'; ExternalVisible := 'False'; ExternalWritable := 'False'; S7_SetPoint := 'False'} : "UDT_Message";   // Message character array
      ss_Status { ExternalAccessible := 'False'; ExternalVisible := 'False'; ExternalWritable := 'False'} : Struct   // Status structure
         FIFOStatus { ExternalAccessible := 'False'; ExternalVisible := 'False'; ExternalWritable := 'False'} : "UDT_FifoStatus";
         FIFOError { ExternalAccessible := 'False'; ExternalVisible := 'False'; ExternalWritable := 'False'; S7_SetPoint := 'True'} : Bool;   // FIFO data buffer full
         FIFOWarning { ExternalAccessible := 'False'; ExternalVisible := 'False'; ExternalWritable := 'False'; S7_SetPoint := 'True'} : Bool;   // FIFO error
         HeartbeatOk { ExternalAccessible := 'False'; ExternalVisible := 'False'; ExternalWritable := 'False'} : Bool;   // FIFO warning
         InvalidTimeInterval { ExternalAccessible := 'False'; ExternalVisible := 'False'; ExternalWritable := 'False'} : Bool;   // Heartbeat ok
         InvalidTimeout { ExternalAccessible := 'False'; ExternalVisible := 'False'; ExternalWritable := 'False'} : Bool;   // Heartbeat time interval lower than zero
         InvalidMsgArraySize { ExternalAccessible := 'False'; ExternalVisible := 'False'; ExternalWritable := 'False'} : Bool;   // Heartbeat timeout lower than zero or lower than heartbeat time interval
      END_STRUCT;
      ss_Message { ExternalAccessible := 'False'; ExternalVisible := 'False'; ExternalWritable := 'False'} : String;   // Message character string
      ss_MSGID { ExternalAccessible := 'False'; ExternalVisible := 'False'; ExternalWritable := 'False'} : String;   // Timestamp
      sui_MsgArrayElNr { ExternalAccessible := 'False'; ExternalVisible := 'False'; ExternalWritable := 'False'} : UInt;   // Invalid message array size
      si_MaxMsgLen { ExternalAccessible := 'False'; ExternalVisible := 'False'; ExternalWritable := 'False'} : Int;   // Maximum message length
      si_MsgLen { ExternalAccessible := 'False'; ExternalVisible := 'False'; ExternalWritable := 'False'} : Int;   // String character message length
      si_LostMsg { ExternalAccessible := 'False'; ExternalVisible := 'False'; ExternalWritable := 'False'} : Int;   // Number of lost messages
      sx_MsgLost { ExternalAccessible := 'False'; ExternalVisible := 'False'; ExternalWritable := 'False'} : Bool;   // Message lost
   END_VAR

   VAR CONSTANT
      cc_NULL : Char := '$00';   // NULL sign
      cs_Start : Char := '$02';   // Termination signs
      cs_End : Char := '$03';
      cs_Length : String := '0006';
      cs_StartOfSort : String := 'SS';   // Message type
   END_VAR


BEGIN
	(*
	----------------------------------------------------------------------------------------

	Version history:
	Date        | Version   | Author        | Remark
	----------------------------------------------------------------------------------------
	24/05/2019  | 0.1       | L.Klar        | first release MHS TIA 15.1
	29/06/2021  | 1.0       | F.Baten       | first release MHS TIA 16.4
	21/02/2023  | 4.0       | F.Baten       | 4.0 Release TIA 17.5
	*)

	REGION 1 – FIFO header status update

	    // Mode 'S' - FIFO register status update
	    "FC_Fifo"(ic_Mode := 'S',
	              qUDT_Status => #ss_Status.FIFOStatus,
	              qx_Error => #ss_Status.FIFOError,
	              qx_Warning => #ss_Status.FIFOWarning,
	              iqv_Data := #s_UDT_MessageArray,
	              iqUDT_FifoHeader := #iqUDT_FifoHeader,
	              iqv_DataBuffer := #iqs_FifoData);


	END_REGION

	REGION 4 – Message preparation

	    #s_R_TRIG_StartOfSort(CLK := #ix_StartOfSort);

	    IF (NOT #iqUDT_FifoHeader.Status.Full)                 // FIFO isn't full
	    THEN

	        IF (#ix_EnableSend                                  // Send is enable
	            AND #s_R_TRIG_StartOfSort.Q                     // Trigger message
	            AND NOT #ss_Status.FIFOError)                   // No FIFO error
	        THEN
	            REGION 4.1 – Message preparation

	                // Heartbeat message composing according to the structure: STX,00,06,SS,ETX
	                #ss_Message := CONCAT(IN1 := #cs_Start,     // Start of message
	                                      IN2 := #cs_Length,    // message length
	                                      IN3 := #cs_StartOfSort,// Start of sort message
	                                      IN4 := #cs_End);      // End of message

	            END_REGION

	            REGION 4.2 – Maximum number of the message characters

	                #si_MaxMsgLen := "FC_GetNrOfArrayEl"(iv_Array := #s_UDT_MessageArray.Character);

	            END_REGION

	            REGION 4.3 – Length of the complete message

	                #si_MsgLen := LEN(#ss_Message);

	            END_REGION

	            REGION 4.4 –  Message array size validation

	                #ss_Status.InvalidMsgArraySize := #si_MsgLen > #si_MaxMsgLen;

	            END_REGION

	            REGION 4.5 –  Message character string conversion to a message array of characters

	                IF (NOT #ss_Status.InvalidMsgArraySize)     // Message character array size is valid
	                THEN

	                    Strg_TO_Chars(Strg := #ss_Message,
	                                  pChars := 0,
	                                  Cnt => #sui_MsgArrayElNr,
	                                  Chars := #s_UDT_MessageArray.Character);

	                END_IF;

	            END_REGION

	            REGION 4.6 – Clearing remaining characters in the message character array

	                IF (NOT #ss_Status.InvalidMsgArraySize)     // Message character array size is valid
	                THEN

	                    // Filling up not used message character array elements with '$00' (ASCII - 16#00)
	                    FILL_BLK(IN := #cc_NULL,
	                             COUNT := UINT_TO_ULINT(INT_TO_UINT(#si_MaxMsgLen) - #sui_MsgArrayElNr),
	                             OUT => #s_UDT_MessageArray.Character[#sui_MsgArrayElNr]);

	                END_IF;

	            END_REGION

	            REGION 4.7 – Message write into a FIFO register

	                IF (#ix_EnableSend                          // Heartbeat send enable
	                    AND NOT #ss_Status.InvalidMsgArraySize) // Message character array size is valid
	                THEN

	                    // Mode 'W' - Write FIFO record
	                    "FC_Fifo"(ic_Mode := 'W',
	                              qUDT_Status => #ss_Status.FIFOStatus,
	                              qx_Error => #ss_Status.FIFOError,
	                              qx_Warning => #ss_Status.FIFOWarning,
	                              iqv_Data := #s_UDT_MessageArray,
	                              iqUDT_FifoHeader := #iqUDT_FifoHeader,
	                              iqv_DataBuffer := #iqs_FifoData);
	                END_IF;

	            END_REGION

	        END_IF;

	        // In case of FIFO full, the FIFO full error bit and FIFO collective error bit are set
	    ELSE

	        #ss_Status.FIFOError := TRUE;
	        #ss_Status.FIFOStatus.FifoFull := TRUE;

	    END_IF;

	END_REGION
END_FUNCTION_BLOCK

FUNCTION_BLOCK "FB_FedExTCPIPReceive"
{ S7_Optimized_Access := 'TRUE' }
VERSION : 0.1
// ATTRIBUTES
// AUTO_NUMBER = True
// BLOCK_NUMBER = 84
// END_ATTRIBUTES
   VAR_INPUT
      iUDT_Connection { ExternalAccessible := 'False'; ExternalVisible := 'False'; ExternalWritable := 'False'} : "UDT_Connection";   // Connection parameters
      ix_EnableReceive { ExternalAccessible := 'False'; ExternalVisible := 'False'; ExternalWritable := 'False'} : Bool;   // TRUE when receive enable
   END_VAR

   VAR_OUTPUT
      qx_Error { ExternalAccessible := 'False'; ExternalVisible := 'False'; ExternalWritable := 'False'} : Bool;   // TRUE when collective block error occurred
      qx_Warning { ExternalAccessible := 'False'; ExternalVisible := 'False'; ExternalWritable := 'False'} : Bool;   // TRUE when collective block warning occurred
   END_VAR

   VAR_IN_OUT
      iqUDT_FifoHeader : "UDT_FifoHeader";   // Fifo header
      iqv_FifoData : Variant;   // Fifo data
      iqUDT_Statistics : "UDT_TCPIPReceiveStatistics";   // Statistic structure
   END_VAR

